// TIA Portal project "examen2" (V15.1)

(* hardware
DEVICE "S7-1200 station_1"  S7-1200 Station
   slot 0: "Rack_0"  S7-1200 Rack  Rack  V1.0
   slot 1: "03_BANDA"  CPU 1212C AC/DC/Rly  6ES7 212-1BE40-0XB0  V4.2
   slot 3: "AQ 1x12BIT_1"  AQ1 signal board  6ES7 232-4HA30-0XB0  V1.0
DEVICE "S7-1200 station_2"  S7-1200 Station
   slot 0: "Rack_0"  S7-1200 Rack  Rack  V1.0
   slot 1: "01_CONTROL"  CPU 1214C AC/DC/Rly  6ES7 214-1BG40-0XB0  V4.2
   slot 2: "DI 8/DQ 8x24VDC_1"  6ES7 223-1BH32-0XB0  V2.0
   slot 3: "AQ 1x12BIT_1"  AQ1 signal board  6ES7 232-4HA30-0XB0  V1.0
DEVICE "S7-1200 station_3"  S7-1200 Station
   slot 0: "Rack_0"  S7-1200 Rack  Rack  V1.0
   slot 1: "02_ALMACEN"  CPU 1214C AC/DC/Rly  6ES7 214-1BG40-0XB0  V4.2
   slot 2: "DI 8x24VDC/DQ 8xRelay_1"  SM 1223 DI8/DQ8 x relay  6ES7 223-1PH32-0XB0  V2.0
*)

// ===== PLC "03_BANDA"  CPU 1212C AC/DC/Rly =====

VAR_GLOBAL   // PLC tag table "Tabla de variables estándar"
   "START" AT %M1.0 : Bool;
   "STOP" AT %M1.1 : Bool;
   "MEM0" AT %M1.2 : Bool;
   "SEN1" AT %I0.3 : Bool;
   "METALCOUNTER" AT %MW10 : Int;
   "PLASTICCOUNTER" AT %MW12 : Int;
   "MEM4" AT %M1.3 : Bool;
   "MEM1" AT %M1.4 : Bool;
   "SEN4" AT %I0.6 : Bool;
   "MEM2" AT %M1.5 : Bool;
   "MEM3" AT %M1.6 : Bool;
   "SEN5" AT %I0.7 : Bool;
   "SEN2" AT %I0.4 : Bool;
   "MEM5" AT %M1.7 : Bool;
   "SEN3" AT %I0.5 : Bool;
   "MOTORBANDA" AT %Q0.0 : Bool;
   "DATARCVS" AT %MB2 : Byte;
   "DATASENDS" AT %MB3 : Byte;
   "Tag_1" AT %QW80 : Int;
   "SUM_ST" AT %MW8 : Int;
   "COUNTER_MEM" AT %M0.0 : Bool;
   "AVISO" AT %M0.1 : Bool;
   "System_Byte" AT %MB1001 : Byte;
   "FirstScan" AT %M1001.0 : Bool;
   "DiagStatusUpdate" AT %M1001.1 : Bool;
   "AlwaysTRUE" AT %M1001.2 : Bool;
   "AlwaysFALSE" AT %M1001.3 : Bool;
   "Clock_Byte" AT %MB1002 : Byte;
   "Clock_10Hz" AT %M1002.0 : Bool;
   "Clock_5Hz" AT %M1002.1 : Bool;
   "Clock_2.5Hz" AT %M1002.2 : Bool;
   "Clock_2Hz" AT %M1002.3 : Bool;
   "Clock_1.25Hz" AT %M1002.4 : Bool;
   "Clock_1Hz" AT %M1002.5 : Bool;
   "Clock_0.625Hz" AT %M1002.6 : Bool;
   "Clock_0.5Hz" AT %M1002.7 : Bool;
   "BYTEINALM" AT %MB4 : Byte;
   "ENDPROCESS" AT %M0.2 : Bool;
   "FIN" AT %M0.3 : Bool;
   "STATUS2SEND" AT %M0.4 : Bool;
   "BYTE2SEND" AT %MB5 : Byte;
   "DATASENDS2" AT %MB6 : Byte;
   "BIT0SUM" AT %M0.5 : Bool;
   "BIT1SUM" AT %M0.6 : Bool;
   "BIT2SUM" AT %M0.7 : Bool;
   "BIT3SUM" AT %M7.0 : Bool;
   "DATA2SENDC" AT %MB14 : Byte;
END_VAR

// folder: System blocks/Program resources

DATA_BLOCK "METALCOUNT"   // DB1
{ S7_Optimized_Access := 'TRUE' }
AUTHOR : Simatic
FAMILY : IEC
NAME : CNTR
VERSION : 1.0
// stored: InstanceOfName IEC_COUNTER
"IEC_COUNTER"
BEGIN
END_DATA_BLOCK

DATA_BLOCK "PLASTCOUNT"   // DB2
{ S7_Optimized_Access := 'TRUE' }
AUTHOR : Simatic
FAMILY : IEC
NAME : CNTR
VERSION : 1.0
// stored: InstanceOfName IEC_COUNTER
"IEC_COUNTER"
BEGIN
END_DATA_BLOCK

DATA_BLOCK "TIM1"   // DB3
{ S7_Optimized_Access := 'TRUE' }
AUTHOR : Simatic
FAMILY : IEC
NAME : IEC_TMR
VERSION : 1.0
// stored: InstanceOfName IEC_TIMER
"IEC_TIMER"
BEGIN
END_DATA_BLOCK

DATA_BLOCK "_03_BANDA_Receive_DB_1"   // DB4
{ S7_Optimized_Access := 'TRUE' }
AUTHOR : SIMATIC
FAMILY : MC7Plus
NAME : TC_IP_v4
VERSION : 1.0
// stored: InstanceOfName TCON_IP_v4
"TCON_IP_v4"
BEGIN
   ID := 1;
   InterfaceId := 64;
   LocalPort := 2000;
   RemoteAddress.ADDR[1] := 192;
   RemoteAddress.ADDR[2] := 168;
   RemoteAddress.ADDR[4] := 2;
END_DATA_BLOCK

DATA_BLOCK "_03_BANDA_Receive_DB"   // DB8
{ S7_Optimized_Access := 'TRUE' }
AUTHOR : SIMATIC
FAMILY : MC7Plus
NAME : TC_IP_v4
VERSION : 1.0
// stored: InstanceOfName TCON_IP_v4
"TCON_IP_v4"
BEGIN
   ID := 3;
   InterfaceId := 64;
   LocalPort := 2001;
   RemoteAddress.ADDR[1] := 192;
   RemoteAddress.ADDR[2] := 168;
   RemoteAddress.ADDR[4] := 1;
END_DATA_BLOCK

DATA_BLOCK "_03_BANDA_Send_DB"   // DB9
{ S7_Optimized_Access := 'TRUE' }
AUTHOR : SIMATIC
FAMILY : MC7Plus
NAME : TC_IP_v4
VERSION : 1.0
// stored: InstanceOfName TCON_IP_v4
"TCON_IP_v4"
BEGIN
   ID := 4;
   InterfaceId := 64;
   RemotePort := 2000;
   ActiveEstablished := true;
   RemoteAddress.ADDR[1] := 192;
   RemoteAddress.ADDR[2] := 168;
   RemoteAddress.ADDR[4] := 1;
END_DATA_BLOCK

DATA_BLOCK "TIMER3"   // DB10
{ S7_Optimized_Access := 'TRUE' }
AUTHOR : Simatic
FAMILY : IEC
NAME : IEC_TMR
VERSION : 1.0
// stored: InstanceOfName IEC_TIMER
"IEC_TIMER"
BEGIN
END_DATA_BLOCK

DATA_BLOCK "_03_BANDA_Send_DB_1"   // DB12
{ S7_Optimized_Access := 'TRUE' }
AUTHOR : SIMATIC
FAMILY : MC7Plus
NAME : TC_IP_v4
VERSION : 1.0
// stored: InstanceOfName TCON_IP_v4
"TCON_IP_v4"
BEGIN
   ID := 2;
   InterfaceId := 64;
   RemotePort := 2000;
   ActiveEstablished := true;
   RemoteAddress.ADDR[1] := 192;
   RemoteAddress.ADDR[2] := 168;
   RemoteAddress.ADDR[4] := 2;
END_DATA_BLOCK

DATA_BLOCK "_03_BANDA_Send_DB_3"   // DB16
{ S7_Optimized_Access := 'TRUE' }
AUTHOR : SIMATIC
FAMILY : MC7Plus
NAME : TC_IP_v4
VERSION : 1.0
// stored: InstanceOfName TCON_IP_v4
"TCON_IP_v4"
BEGIN
   ID := 6;
   InterfaceId := 64;
   RemotePort := 2002;
   ActiveEstablished := true;
   RemoteAddress.ADDR[1] := 192;
   RemoteAddress.ADDR[2] := 168;
   RemoteAddress.ADDR[4] := 1;
END_DATA_BLOCK

DATA_BLOCK "_03_BANDA_Send_DB_2"   // DB18
{ S7_Optimized_Access := 'TRUE' }
AUTHOR : SIMATIC
FAMILY : MC7Plus
NAME : TC_IP_v4
VERSION : 1.0
// stored: InstanceOfName TCON_IP_v4
"TCON_IP_v4"
BEGIN
   ID := 5;
   InterfaceId := 64;
   RemotePort := 2000;
   ActiveEstablished := true;
   RemoteAddress.ADDR[1] := 192;
   RemoteAddress.ADDR[2] := 168;
   RemoteAddress.ADDR[4] := 1;
END_DATA_BLOCK

// folder: (top level)

FUNCTION "CODER" : Void   // FC1, FBD
{ S7_Optimized_Access := 'TRUE' }
VERSION : 0.1
   VAR_INPUT
      BIT0 : Bool;
      BIT1 : Bool;
      BIT2 : Bool;
      BIT3 : Bool;
      BIT4 : Bool;
      BIT5 : Bool;
      BIT6 : Bool;
      BIT7 : Bool;
   END_VAR
   VAR_IN_OUT
      OUT : Byte;
   END_VAR
   VAR_TEMP
      MASK0 : Byte;
      MASK1 : Byte;
      MASK2 : Byte;
      MASK3 : Byte;
      MASK4 : Byte;
      MASK5 : Byte;
      MASK6 : Byte;
      MASK7 : Byte;
      MASK : Byte;
      MASK0N : Byte;
      MASK1N : Byte;
      MASK2N : Byte;
      MASK3N : Byte;
      MASK4N : Byte;
      MASK5N : Byte;
      MASK6N : Byte;
      MASK7N : Byte;
      MASKN : Byte;
   END_VAR
BEGIN

REGION Network 1
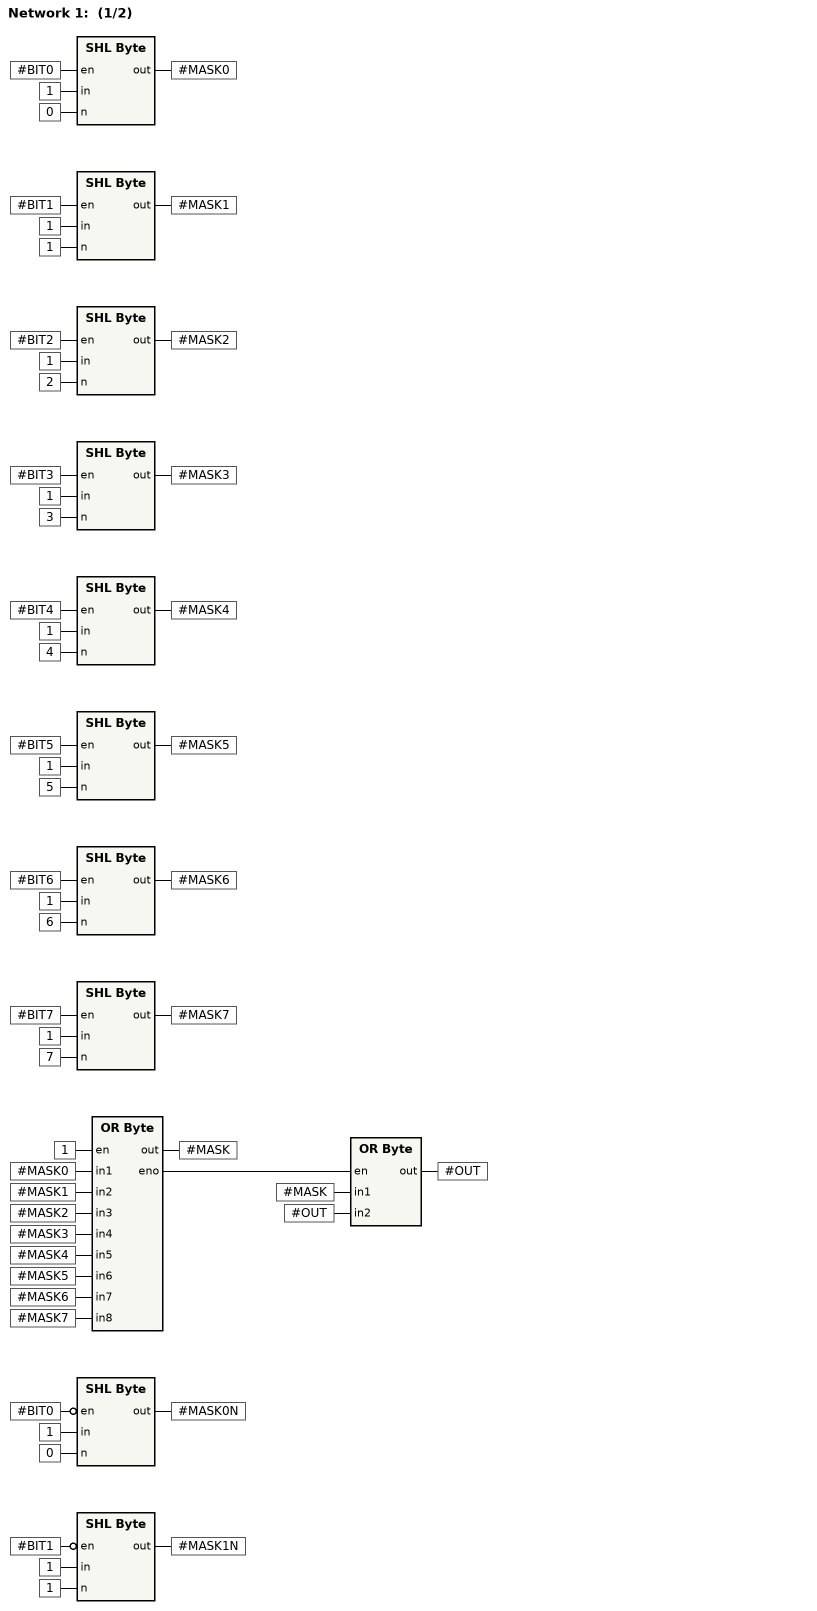
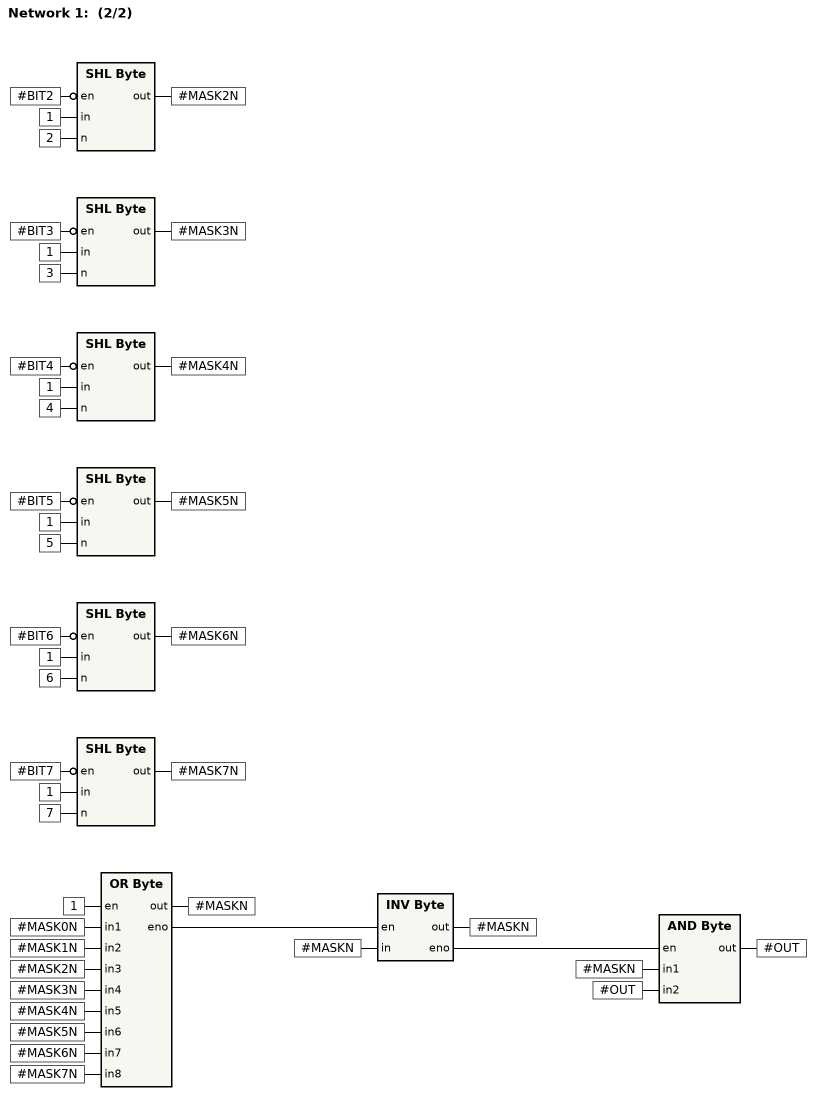
   IF #BIT0 THEN #MASK0 := SHL(IN := 1, N := 0); END_IF;
   IF #BIT1 THEN #MASK1 := SHL(IN := 1, N := 1); END_IF;
   IF #BIT2 THEN #MASK2 := SHL(IN := 1, N := 2); END_IF;
   IF #BIT3 THEN #MASK3 := SHL(IN := 1, N := 3); END_IF;
   IF #BIT4 THEN #MASK4 := SHL(IN := 1, N := 4); END_IF;
   IF #BIT5 THEN #MASK5 := SHL(IN := 1, N := 5); END_IF;
   IF #BIT6 THEN #MASK6 := SHL(IN := 1, N := 6); END_IF;
   IF #BIT7 THEN #MASK7 := SHL(IN := 1, N := 7); END_IF;
   IF 1 THEN
       #MASK := #MASK0 OR #MASK1 OR #MASK2 OR #MASK3 OR #MASK4 OR #MASK5 OR #MASK6 OR #MASK7;
       #OUT := #MASK OR #OUT;
   END_IF;
   IF NOT #BIT0 THEN #MASK0N := SHL(IN := 1, N := 0); END_IF;
   IF NOT #BIT1 THEN #MASK1N := SHL(IN := 1, N := 1); END_IF;
   IF NOT #BIT2 THEN #MASK2N := SHL(IN := 1, N := 2); END_IF;
   IF NOT #BIT3 THEN #MASK3N := SHL(IN := 1, N := 3); END_IF;
   IF NOT #BIT4 THEN #MASK4N := SHL(IN := 1, N := 4); END_IF;
   IF NOT #BIT5 THEN #MASK5N := SHL(IN := 1, N := 5); END_IF;
   IF NOT #BIT6 THEN #MASK6N := SHL(IN := 1, N := 6); END_IF;
   IF NOT #BIT7 THEN #MASK7N := SHL(IN := 1, N := 7); END_IF;
   IF 1 THEN
       #MASKN := #MASK0N OR #MASK1N OR #MASK2N OR #MASK3N OR #MASK4N OR #MASK5N OR #MASK6N OR #MASK7N;
       #MASKN := NOT #MASKN;
       #OUT := #MASKN AND #OUT;
   END_IF;
END_REGION
END_FUNCTION

FUNCTION "DECODER" : Void   // FC2, FBD
{ S7_Optimized_Access := 'TRUE' }
VERSION : 0.1
   VAR_INPUT
      INBYTE : Byte;
   END_VAR
   VAR_OUTPUT
      BIT0 : Bool;
      BIT1 : Bool;
      BIT2 : Bool;
      BIT3 : Bool;
      BIT4 : Bool;
      BIT5 : Bool;
      BIT6 : Bool;
      BIT7 : Bool;
   END_VAR
   VAR_TEMP
      MASK0 : Byte;
      MASK1 : Byte;
      MASK2 : Byte;
      MASK3 : Byte;
      MASK4 : Byte;
      MASK5 : Byte;
      MASK6 : Byte;
      MASK7 : Byte;
      OUTBIT0 : Byte;
      OUTBIT1 : Byte;
      OUTBIT2 : Byte;
      OUTBIT3 : Byte;
      OUTBIT4 : Byte;
      OUTBIT5 : Byte;
      OUTBIT6 : Byte;
      OUTBIT7 : Byte;
   END_VAR
BEGIN

REGION Network 1
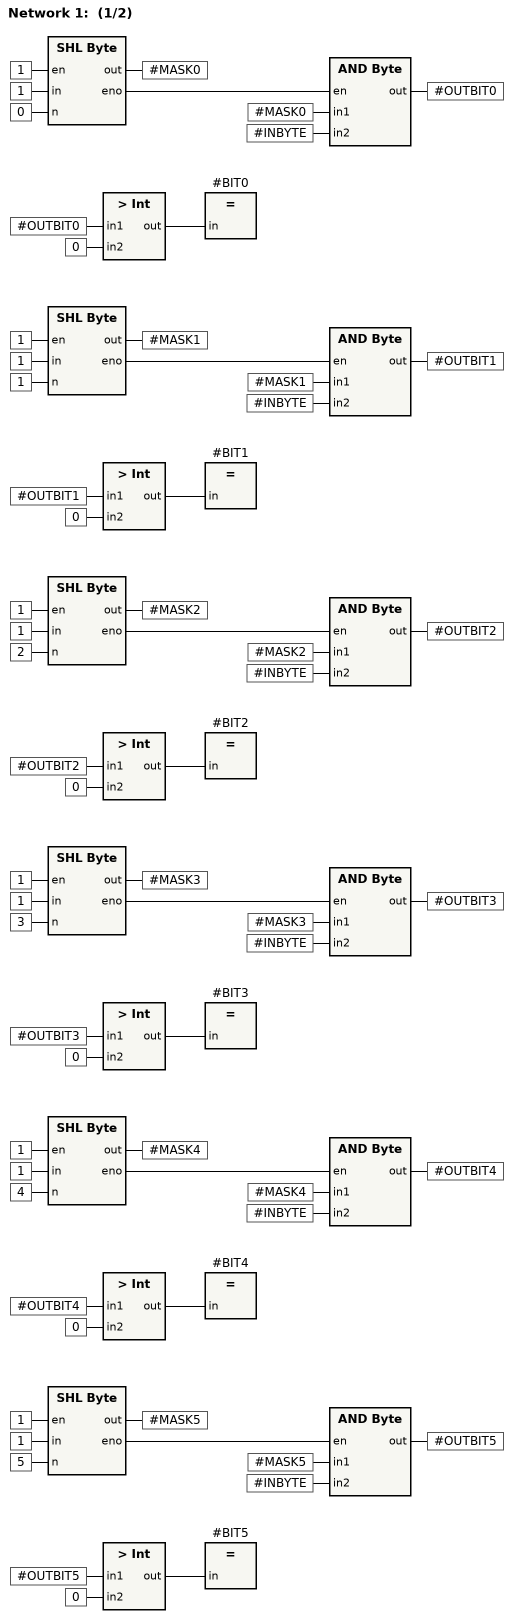
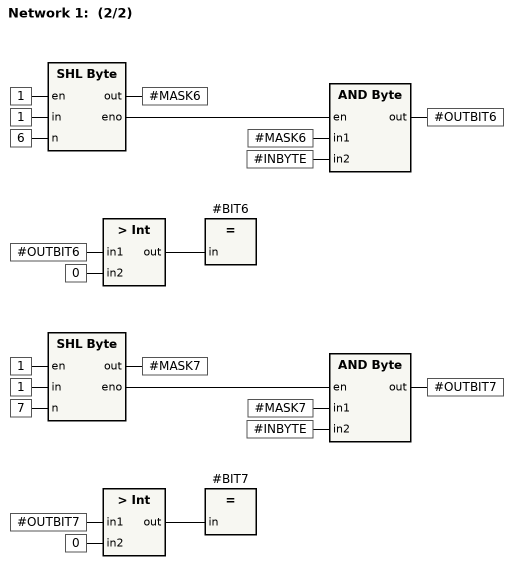
   IF 1 THEN
       #MASK0 := SHL(IN := 1, N := 0);
       #OUTBIT0 := #MASK0 AND #INBYTE;
   END_IF;
   #BIT0 := #OUTBIT0 > 0;
   IF 1 THEN
       #MASK1 := SHL(IN := 1, N := 1);
       #OUTBIT1 := #MASK1 AND #INBYTE;
   END_IF;
   #BIT1 := #OUTBIT1 > 0;
   IF 1 THEN
       #MASK2 := SHL(IN := 1, N := 2);
       #OUTBIT2 := #MASK2 AND #INBYTE;
   END_IF;
   #BIT2 := #OUTBIT2 > 0;
   IF 1 THEN
       #MASK3 := SHL(IN := 1, N := 3);
       #OUTBIT3 := #MASK3 AND #INBYTE;
   END_IF;
   #BIT3 := #OUTBIT3 > 0;
   IF 1 THEN
       #MASK4 := SHL(IN := 1, N := 4);
       #OUTBIT4 := #MASK4 AND #INBYTE;
   END_IF;
   #BIT4 := #OUTBIT4 > 0;
   IF 1 THEN
       #MASK5 := SHL(IN := 1, N := 5);
       #OUTBIT5 := #MASK5 AND #INBYTE;
   END_IF;
   #BIT5 := #OUTBIT5 > 0;
   IF 1 THEN
       #MASK6 := SHL(IN := 1, N := 6);
       #OUTBIT6 := #MASK6 AND #INBYTE;
   END_IF;
   #BIT6 := #OUTBIT6 > 0;
   IF 1 THEN
       #MASK7 := SHL(IN := 1, N := 7);
       #OUTBIT7 := #MASK7 AND #INBYTE;
   END_IF;
   #BIT7 := #OUTBIT7 > 0;
END_REGION
END_FUNCTION

FUNCTION "DecToBin" : Void   // FC3, FBD
{ S7_Optimized_Access := 'TRUE' }
VERSION : 0.1
   VAR_INPUT
      dec : Int;
   END_VAR
   VAR_OUTPUT
      bit0 : Bool;
      bit1 : Bool;
      bit2 : Bool;
      bit3 : Bool;
   END_VAR
   VAR_TEMP
      secdec : Int;
      thirdec : Int;
      quardec : Int;
      bit0s : Int;
      bit1s : Int;
      bit2s : Int;
      bit3s : Int;
   END_VAR
BEGIN

REGION Network 1
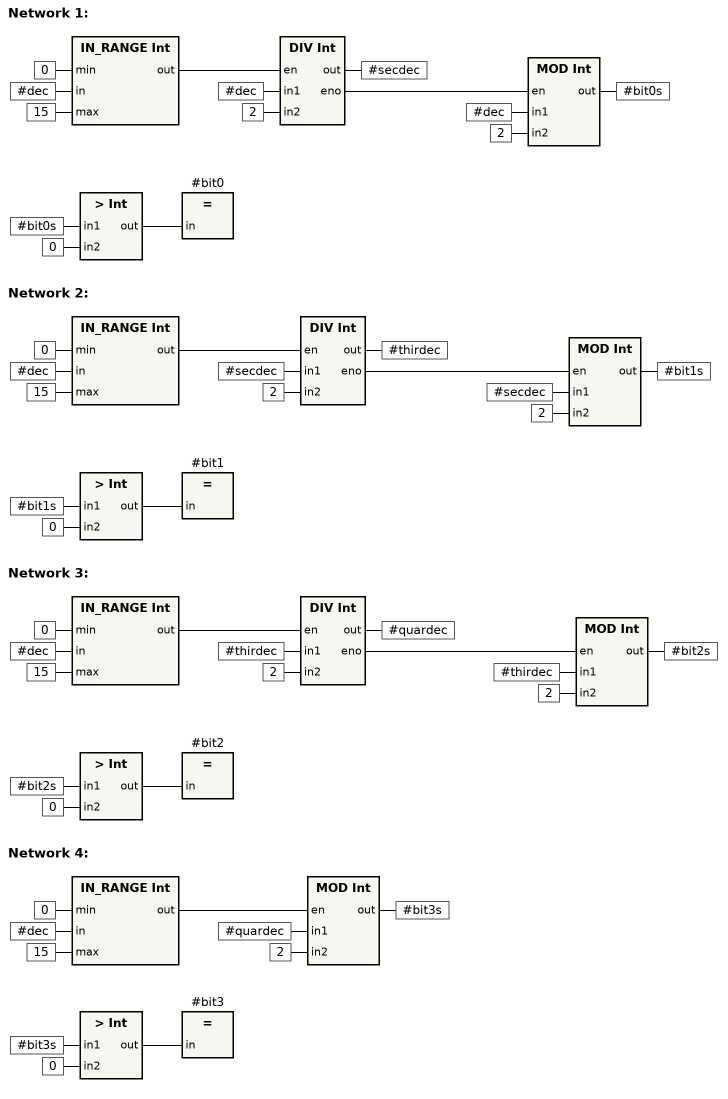
   IF (0 <= #dec) AND (#dec <= 15) THEN
       #secdec := #dec / 2;
       #bit0s := #dec MOD 2;
   END_IF;
   #bit0 := #bit0s > 0;
END_REGION

REGION Network 2
   IF (0 <= #dec) AND (#dec <= 15) THEN
       #thirdec := #secdec / 2;
       #bit1s := #secdec MOD 2;
   END_IF;
   #bit1 := #bit1s > 0;
END_REGION

REGION Network 3
   IF (0 <= #dec) AND (#dec <= 15) THEN
       #quardec := #thirdec / 2;
       #bit2s := #thirdec MOD 2;
   END_IF;
   #bit2 := #bit2s > 0;
END_REGION

REGION Network 4
   IF (0 <= #dec) AND (#dec <= 15) THEN #bit3s := #quardec MOD 2; END_IF;
   #bit3 := #bit3s > 0;
END_REGION
END_FUNCTION

FUNCTION "BinToDec" : Void   // FC4, FBD
{ S7_Optimized_Access := 'TRUE' }
VERSION : 0.1
   VAR_INPUT
      bit0 : Bool;
      bit1 : Bool;
      bit2 : Bool;
      bit3 : Bool;
   END_VAR
   VAR_OUTPUT
      decimal : Int;
   END_VAR
   VAR_TEMP
      dec0 : Int;
      dec1 : Int;
      dec2 : Int;
      dec3 : Int;
   END_VAR
BEGIN

REGION Network 1
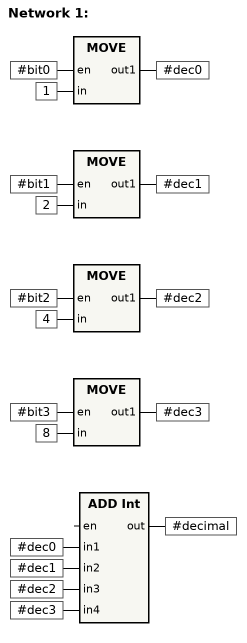
   IF #bit0 THEN #dec0 := 1; END_IF;
   IF #bit1 THEN #dec1 := 2; END_IF;
   IF #bit2 THEN #dec2 := 4; END_IF;
   IF #bit3 THEN #dec3 := 8; END_IF;
   #decimal := #dec0 + #dec1 + #dec2 + #dec3;
END_REGION
END_FUNCTION

ORGANIZATION_BLOCK "Main"   // OB1, LAD, ProgramCycle
TITLE = "Main Program Sweep (Cycle)" / "SLAVE_CONVEYOR_PLC"
{ S7_Optimized_Access := 'TRUE' }
VERSION : 0.1
   VAR_INPUT
      Initial_Call : Bool;   // Initial call of this OB
      Remanence : Bool;   // =True, if remanent data are available
   END_VAR
   VAR_TEMP
      SUMA : DInt;
      SUMA_ : Int;
      SUM_ : Int;
      BIT2 : Bool;
      BIT5 : Bool;
      BIT4 : Bool;
      BIT6 : Bool;
      BIT3 : Bool;
      BIT7 : Bool;
      MEM6 : Bool;
      MBIT0 : Bool;
      MBIT1 : Bool;
      MBIT2 : Bool;
      MBIT3 : Bool;
      MBIT4 : Bool;
      MBIT5 : Bool;
      MBIT6 : Bool;
   END_VAR
   VAR_TEMP   // added for the SCL form of the ladder/FBD networks
      _w1 : Bool;
   END_VAR
BEGIN

REGION Network 1: LOGIC_SEGMENT
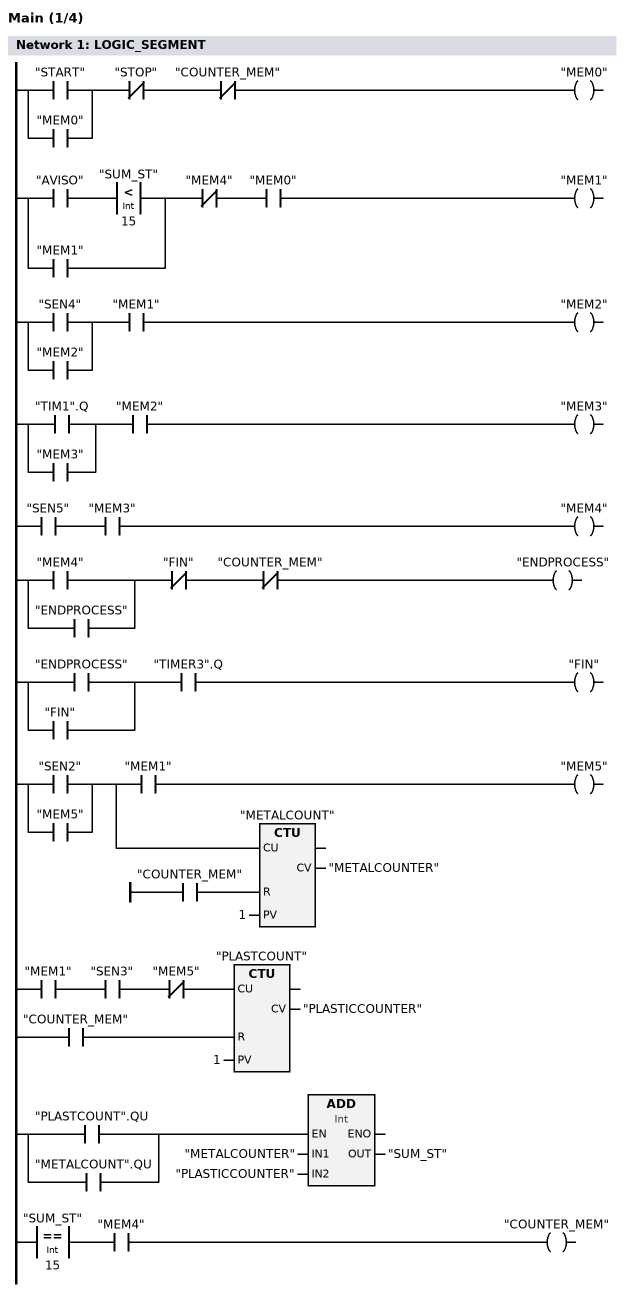
   "MEM0" := ("START" OR "MEM0") AND NOT "STOP" AND NOT "COUNTER_MEM";
   "MEM1" := (("AVISO" AND ("SUM_ST" < 15)) OR "MEM1") AND NOT "MEM4" AND "MEM0";
   "MEM2" := ("SEN4" OR "MEM2") AND "MEM1";
   "MEM3" := ("TIM1".Q OR "MEM3") AND "MEM2";
   "MEM4" := "SEN5" AND "MEM3";
   "ENDPROCESS" := ("MEM4" OR "ENDPROCESS") AND NOT "FIN" AND NOT "COUNTER_MEM";
   "FIN" := ("ENDPROCESS" OR "FIN") AND "TIMER3".Q;
   #_w1 := "SEN2" OR "MEM5";
   "MEM5" := #_w1 AND "MEM1";
   "METALCOUNT".CTU(CU := #_w1, R := "COUNTER_MEM", PV := 1, CV => "METALCOUNTER");
   "PLASTCOUNT".CTU(CU := "MEM1" AND "SEN3" AND NOT "MEM5", R := "COUNTER_MEM", PV := 1, CV => "PLASTICCOUNTER");
   IF "PLASTCOUNT".QU OR "METALCOUNT".QU THEN "SUM_ST" := "METALCOUNTER" + "PLASTICCOUNTER"; END_IF;
   "COUNTER_MEM" := ("SUM_ST" = 15) AND "MEM4";
END_REGION

REGION Network 2: MECHANICAL_SEGMENT
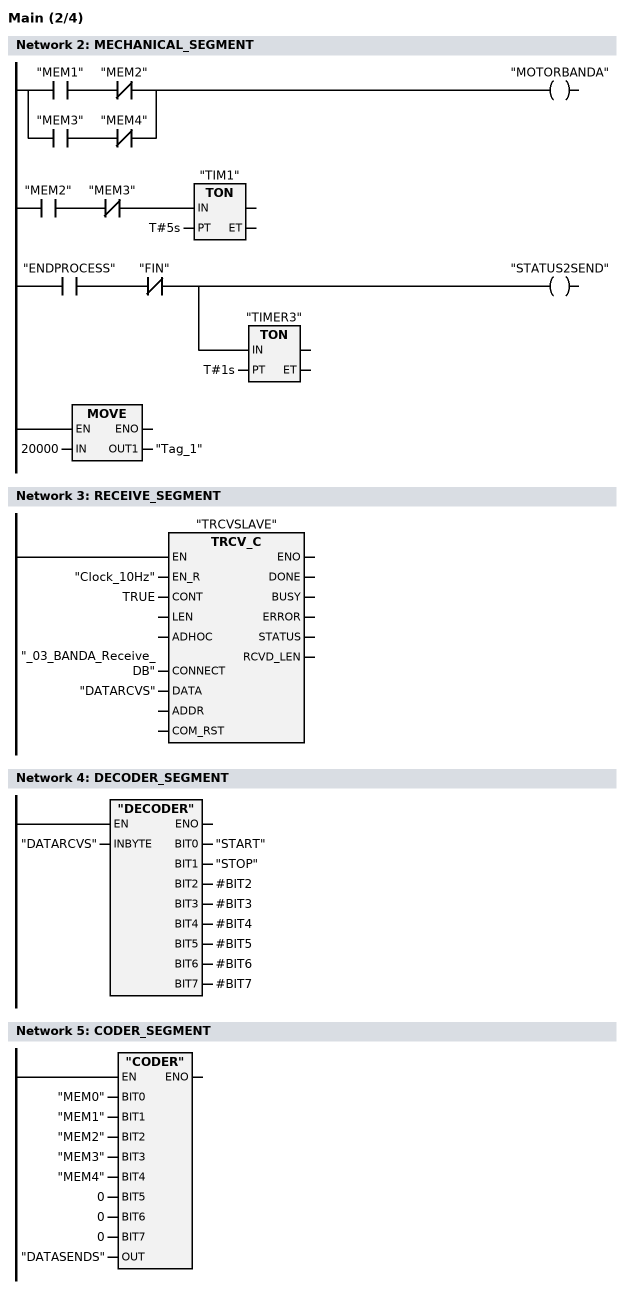
   "MOTORBANDA" := ("MEM1" AND NOT "MEM2") OR ("MEM3" AND NOT "MEM4");
   "TIM1".TON(IN := "MEM2" AND NOT "MEM3", PT := T#5s);
   "STATUS2SEND" := "ENDPROCESS" AND NOT "FIN";
   "TIMER3".TON(IN := "STATUS2SEND", PT := T#1s);
   "Tag_1" := 20000;
END_REGION

REGION Network 3: RECEIVE_SEGMENT
   "TRCVSLAVE"(EN_R := "Clock_10Hz", CONT := TRUE, CONNECT := "_03_BANDA_Receive_DB", DATA := "DATARCVS");   // TRCV_C
END_REGION

REGION Network 4: DECODER_SEGMENT
   RUNG wire#powerrail
      "DECODER"(INBYTE := "DATARCVS", BIT0 => "START", BIT1 => "STOP", BIT2 => #BIT2, BIT3 => #BIT3, BIT4 => #BIT4, BIT5 => #BIT5, BIT6 => #BIT6, BIT7 => #BIT7)
   END_RUNG
   // the same network as SCL:
   "DECODER"(INBYTE := "DATARCVS",
             BIT0 => "START",
             BIT1 => "STOP",
             BIT2 => #BIT2,
             BIT3 => #BIT3,
             BIT4 => #BIT4,
             BIT5 => #BIT5,
             BIT6 => #BIT6,
             BIT7 => #BIT7);
END_REGION

REGION Network 5: CODER_SEGMENT
   RUNG wire#powerrail
      "CODER"(BIT0 := "MEM0", BIT1 := "MEM1", BIT2 := "MEM2", BIT3 := "MEM3", BIT4 := "MEM4", BIT5 := 0, BIT6 := 0, BIT7 := 0, OUT := "DATASENDS")
   END_RUNG
   // the same network as SCL:
   "CODER"(BIT0 := "MEM0",
           BIT1 := "MEM1",
           BIT2 := "MEM2",
           BIT3 := "MEM3",
           BIT4 := "MEM4",
           BIT5 := 0,
           BIT6 := 0,
           BIT7 := 0,
           OUT := "DATASENDS");
END_REGION

REGION Network 6: SEND_SEGMENT
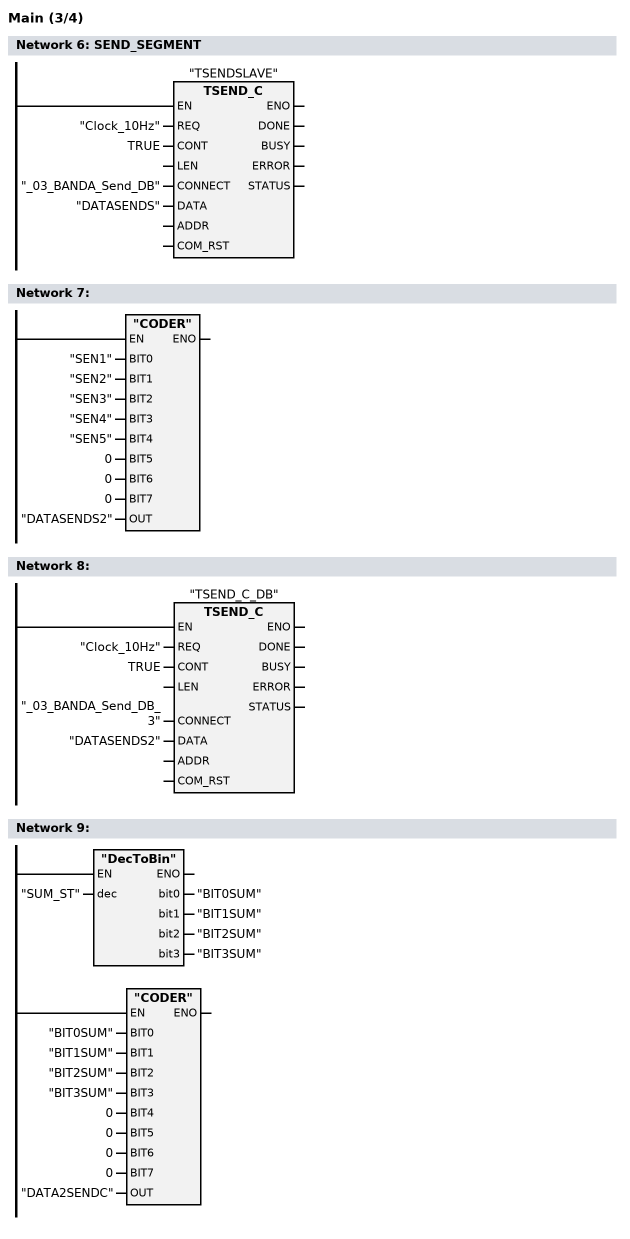
   "TSENDSLAVE"(REQ := "Clock_10Hz", CONT := TRUE, CONNECT := "_03_BANDA_Send_DB", DATA := "DATASENDS");   // TSEND_C
END_REGION

REGION Network 7
   RUNG wire#powerrail
      "CODER"(BIT0 := "SEN1", BIT1 := "SEN2", BIT2 := "SEN3", BIT3 := "SEN4", BIT4 := "SEN5", BIT5 := 0, BIT6 := 0, BIT7 := 0, OUT := "DATASENDS2")
   END_RUNG
   // the same network as SCL:
   "CODER"(BIT0 := "SEN1",
           BIT1 := "SEN2",
           BIT2 := "SEN3",
           BIT3 := "SEN4",
           BIT4 := "SEN5",
           BIT5 := 0,
           BIT6 := 0,
           BIT7 := 0,
           OUT := "DATASENDS2");
END_REGION

REGION Network 8
   "TSEND_C_DB"(REQ := "Clock_10Hz", CONT := TRUE, CONNECT := "_03_BANDA_Send_DB_3", DATA := "DATASENDS2");   // TSEND_C
END_REGION

REGION Network 9
   RUNG wire#powerrail
      "DecToBin"(dec := "SUM_ST", bit0 => "BIT0SUM", bit1 => "BIT1SUM", bit2 => "BIT2SUM", bit3 => "BIT3SUM")
   END_RUNG
   RUNG wire#powerrail
      "CODER"(BIT0 := "BIT0SUM", BIT1 := "BIT1SUM", BIT2 := "BIT2SUM", BIT3 := "BIT3SUM", BIT4 := 0, BIT5 := 0, BIT6 := 0, BIT7 := 0, OUT := "DATA2SENDC")
   END_RUNG
   // the same network as SCL:
   "DecToBin"(dec := "SUM_ST", bit0 => "BIT0SUM", bit1 => "BIT1SUM", bit2 => "BIT2SUM", bit3 => "BIT3SUM");
   "CODER"(BIT0 := "BIT0SUM",
           BIT1 := "BIT1SUM",
           BIT2 := "BIT2SUM",
           BIT3 := "BIT3SUM",
           BIT4 := 0,
           BIT5 := 0,
           BIT6 := 0,
           BIT7 := 0,
           OUT := "DATA2SENDC");
END_REGION

REGION Network 10
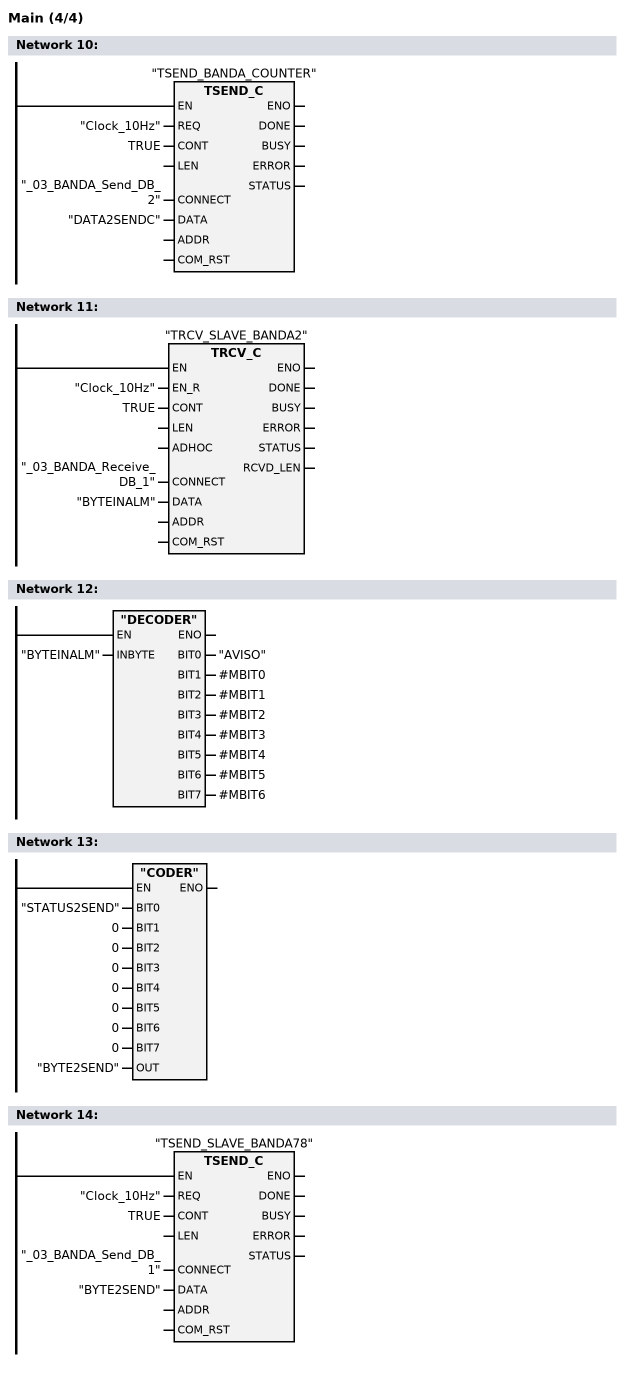
   "TSEND_BANDA_COUNTER"(REQ := "Clock_10Hz",   // TSEND_C
                         CONT := TRUE,
                         CONNECT := "_03_BANDA_Send_DB_2",
                         DATA := "DATA2SENDC");
END_REGION

REGION Network 11
   "TRCV_SLAVE_BANDA2"(EN_R := "Clock_10Hz",   // TRCV_C
                       CONT := TRUE,
                       CONNECT := "_03_BANDA_Receive_DB_1",
                       DATA := "BYTEINALM");
END_REGION

REGION Network 12
   RUNG wire#powerrail
      "DECODER"(INBYTE := "BYTEINALM", BIT0 => "AVISO", BIT1 => #MBIT0, BIT2 => #MBIT1, BIT3 => #MBIT2, BIT4 => #MBIT3, BIT5 => #MBIT4, BIT6 => #MBIT5, BIT7 => #MBIT6)
   END_RUNG
   // the same network as SCL:
   "DECODER"(INBYTE := "BYTEINALM",
             BIT0 => "AVISO",
             BIT1 => #MBIT0,
             BIT2 => #MBIT1,
             BIT3 => #MBIT2,
             BIT4 => #MBIT3,
             BIT5 => #MBIT4,
             BIT6 => #MBIT5,
             BIT7 => #MBIT6);
END_REGION

REGION Network 13
   RUNG wire#powerrail
      "CODER"(BIT0 := "STATUS2SEND", BIT1 := 0, BIT2 := 0, BIT3 := 0, BIT4 := 0, BIT5 := 0, BIT6 := 0, BIT7 := 0, OUT := "BYTE2SEND")
   END_RUNG
   // the same network as SCL:
   "CODER"(BIT0 := "STATUS2SEND",
           BIT1 := 0,
           BIT2 := 0,
           BIT3 := 0,
           BIT4 := 0,
           BIT5 := 0,
           BIT6 := 0,
           BIT7 := 0,
           OUT := "BYTE2SEND");
END_REGION

REGION Network 14
   "TSEND_SLAVE_BANDA78"(REQ := "Clock_10Hz",   // TSEND_C
                         CONT := TRUE,
                         CONNECT := "_03_BANDA_Send_DB_1",
                         DATA := "BYTE2SEND");
END_REGION
END_ORGANIZATION_BLOCK

// ===== PLC "01_CONTROL"  CPU 1214C AC/DC/Rly =====

VAR_GLOBAL   // PLC tag table "Tabla de variables estándar"
   "START" AT %I0.0 : Bool;
   "STOP" AT %I0.1 : Bool;
   "MEM0" AT %M1.0 : Bool;
   "DATASENDM" AT %MB1 : Byte;
   "MEM1" AT %M1.2 : Bool;
   "MEM2" AT %M1.3 : Bool;
   "GREEN" AT %Q8.5 : Bool;
   "MEM3" AT %M1.4 : Bool;
   "MEM4" AT %M1.5 : Bool;
   "ORANGE" AT %Q8.6 : Bool;
   "RED" AT %Q8.7 : Bool;
   "DATARCVM" AT %MB2 : Byte;
   "START2" AT %M3.0 : Bool;
   "SEN1" AT %M1.7 : Bool;
   "STOP2" AT %M0.0 : Bool;
   "TRY" AT %Q0.0 : Bool;
   "System_Byte" AT %MB10 : Byte;
   "FirstScan" AT %M10.0 : Bool;
   "DiagStatusUpdate" AT %M10.1 : Bool;
   "AlwaysTRUE" AT %M10.2 : Bool;
   "AlwaysFALSE" AT %M10.3 : Bool;
   "Clock_Byte" AT %MB11 : Byte;
   "Clock_10Hz" AT %M11.0 : Bool;
   "Clock_5Hz" AT %M11.1 : Bool;
   "Clock_2.5Hz" AT %M11.2 : Bool;
   "Clock_2Hz" AT %M11.3 : Bool;
   "Clock_1.25Hz" AT %M11.4 : Bool;
   "Clock_1Hz" AT %M11.5 : Bool;
   "Clock_0.625Hz" AT %M11.6 : Bool;
   "Clock_0.5Hz" AT %M11.7 : Bool;
   "SEN4" AT %M0.1 : Bool;
   "SEN3" AT %M0.2 : Bool;
   "SEN2" AT %M0.3 : Bool;
   "SEN5" AT %M0.4 : Bool;
   "COUNT1" AT %MB7 : Byte;
   "DATARCVS" AT %MB6 : Byte;
END_VAR

DATA_BLOCK "Data_block_1"   // DB2
{ S7_Optimized_Access := 'FALSE' }
VERSION : 0.1
   VAR
      BYTE0 : Byte;
      BYTE1 : Byte;
      BYTE2 : Byte;
      BYTE4 : Byte;
   END_VAR
BEGIN
END_DATA_BLOCK

// folder: System blocks/Program resources

DATA_BLOCK "_01_CONTROL_Receive_DB_1"   // DB3
{ S7_Optimized_Access := 'TRUE' }
AUTHOR : SIMATIC
FAMILY : MC7Plus
NAME : TC_IP_v4
VERSION : 1.0
// stored: InstanceOfName TCON_IP_v4
"TCON_IP_v4"
BEGIN
   ID := 1;
   InterfaceId := 64;
   LocalPort := 2000;
   RemoteAddress.ADDR[1] := 192;
   RemoteAddress.ADDR[2] := 168;
   RemoteAddress.ADDR[4] := 3;
END_DATA_BLOCK

DATA_BLOCK "_01_CONTROL_Send_DB"   // DB5
{ S7_Optimized_Access := 'TRUE' }
AUTHOR : SIMATIC
FAMILY : MC7Plus
NAME : TC_IP_v4
VERSION : 1.0
// stored: InstanceOfName TCON_IP_v4
"TCON_IP_v4"
BEGIN
   ID := 3;
   InterfaceId := 64;
   RemotePort := 2001;
   ActiveEstablished := true;
   RemoteAddress.ADDR[1] := 192;
   RemoteAddress.ADDR[2] := 168;
   RemoteAddress.ADDR[4] := 3;
END_DATA_BLOCK

DATA_BLOCK "_01_CONTROL_Receive_DB"   // DB6
{ S7_Optimized_Access := 'TRUE' }
AUTHOR : SIMATIC
FAMILY : MC7Plus
NAME : TC_IP_v4
VERSION : 1.0
// stored: InstanceOfName TCON_IP_v4
"TCON_IP_v4"
BEGIN
   ID := 4;
   InterfaceId := 64;
   LocalPort := 2000;
   RemoteAddress.ADDR[1] := 192;
   RemoteAddress.ADDR[2] := 168;
   RemoteAddress.ADDR[4] := 3;
END_DATA_BLOCK

DATA_BLOCK "_01_CONTROL_Receive_DB_2"   // DB7
{ S7_Optimized_Access := 'TRUE' }
AUTHOR : SIMATIC
FAMILY : MC7Plus
NAME : TC_IP_v4
VERSION : 1.0
// stored: InstanceOfName TCON_IP_v4
"TCON_IP_v4"
BEGIN
   ID := 2;
   InterfaceId := 64;
   LocalPort := 2002;
   RemoteAddress.ADDR[1] := 192;
   RemoteAddress.ADDR[2] := 168;
   RemoteAddress.ADDR[4] := 3;
END_DATA_BLOCK

// folder: (top level)

FUNCTION "CODER" : Void   // FC1, FBD
{ S7_Optimized_Access := 'TRUE' }
VERSION : 0.1
   VAR_INPUT
      BIT0 : Bool;
      BIT1 : Bool;
      BIT2 : Bool;
      BIT3 : Bool;
      BIT4 : Bool;
      BIT5 : Bool;
      BIT6 : Bool;
      BIT7 : Bool;
   END_VAR
   VAR_IN_OUT
      OUT : Byte;
   END_VAR
   VAR_TEMP
      MASK0 : Byte;
      MASK1 : Byte;
      MASK2 : Byte;
      MASK3 : Byte;
      MASK4 : Byte;
      MASK5 : Byte;
      MASK6 : Byte;
      MASK7 : Byte;
      MASK : Byte;
      MASK0N : Byte;
      MASK1N : Byte;
      MASK2N : Byte;
      MASK3N : Byte;
      MASK4N : Byte;
      MASK5N : Byte;
      MASK6N : Byte;
      MASK7N : Byte;
      MASKN : Byte;
   END_VAR
BEGIN

REGION Network 1
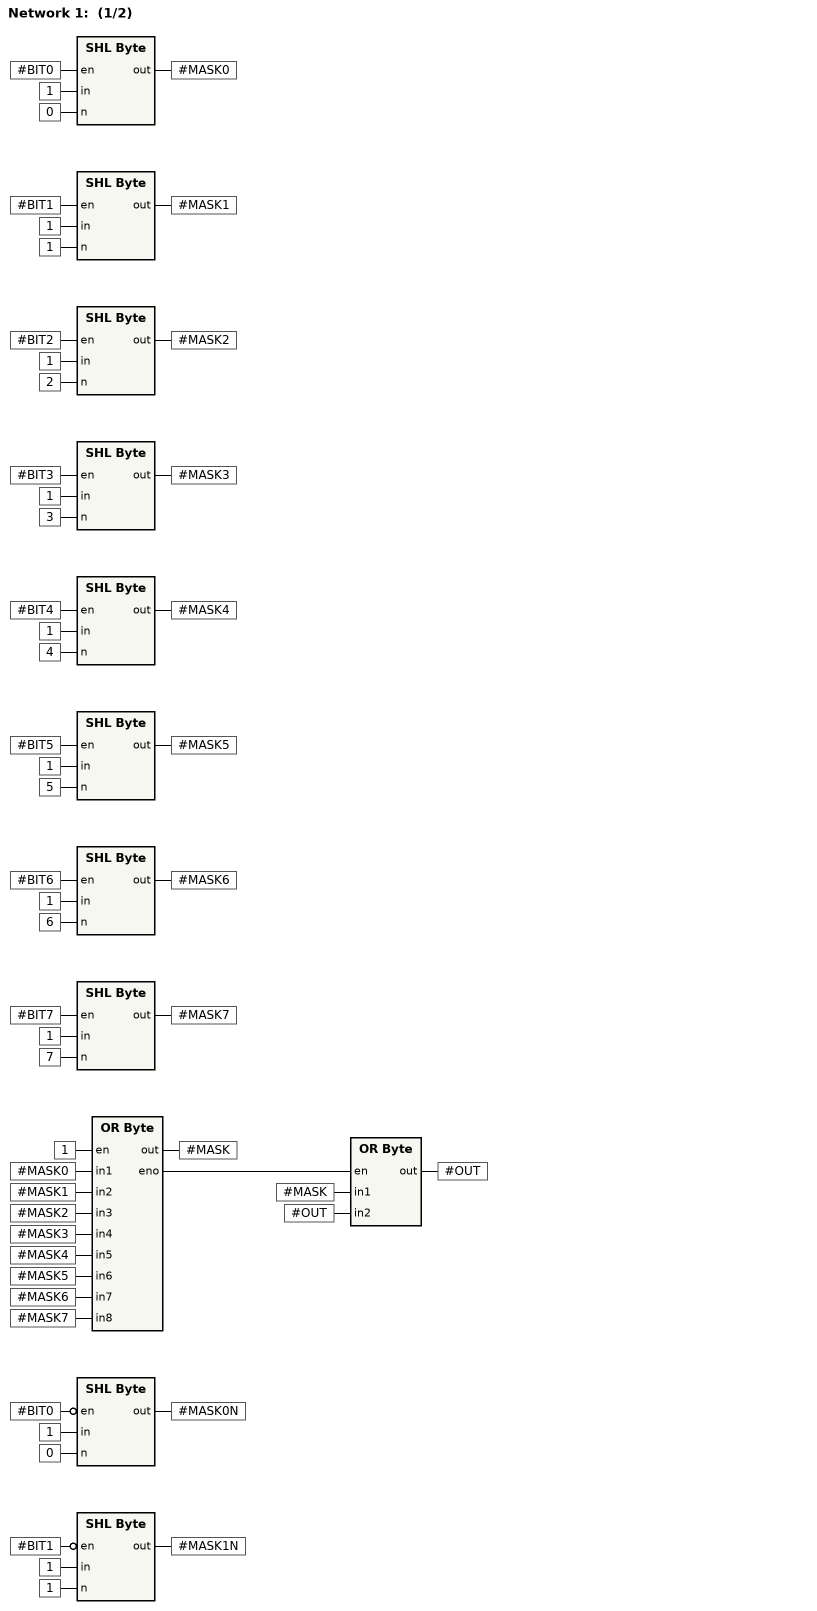
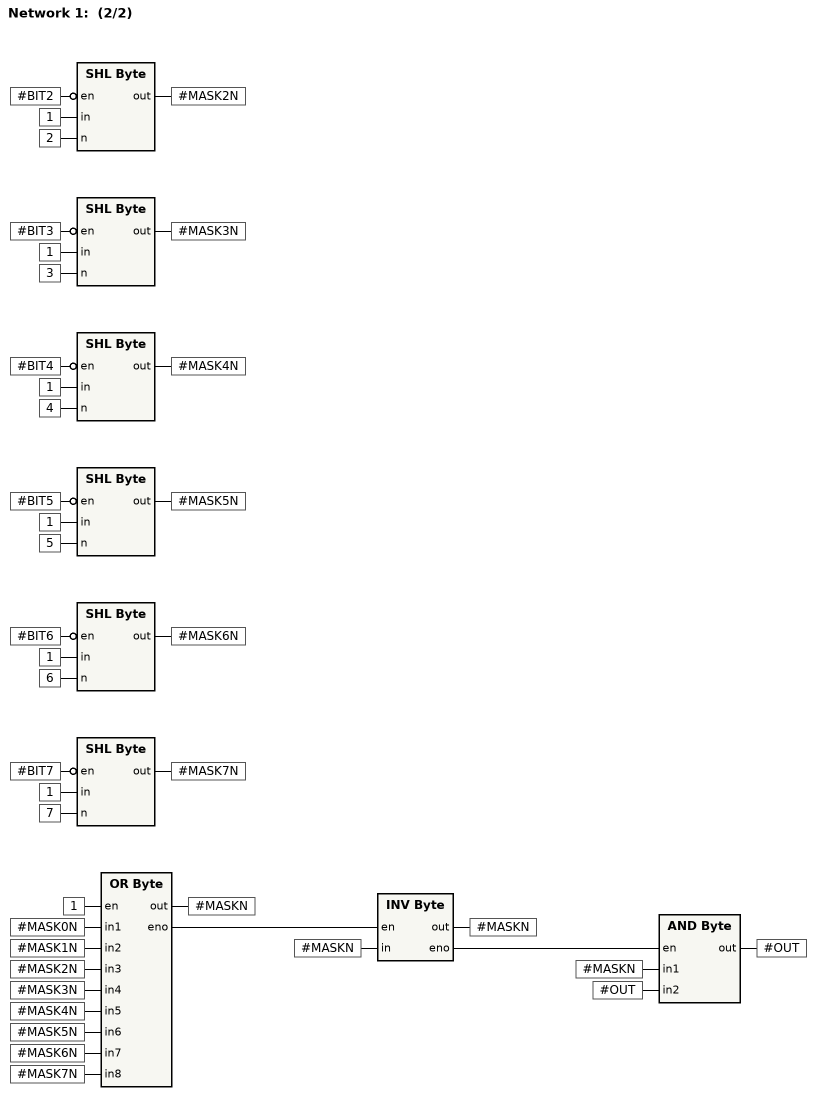
   IF #BIT0 THEN #MASK0 := SHL(IN := 1, N := 0); END_IF;
   IF #BIT1 THEN #MASK1 := SHL(IN := 1, N := 1); END_IF;
   IF #BIT2 THEN #MASK2 := SHL(IN := 1, N := 2); END_IF;
   IF #BIT3 THEN #MASK3 := SHL(IN := 1, N := 3); END_IF;
   IF #BIT4 THEN #MASK4 := SHL(IN := 1, N := 4); END_IF;
   IF #BIT5 THEN #MASK5 := SHL(IN := 1, N := 5); END_IF;
   IF #BIT6 THEN #MASK6 := SHL(IN := 1, N := 6); END_IF;
   IF #BIT7 THEN #MASK7 := SHL(IN := 1, N := 7); END_IF;
   IF 1 THEN
       #MASK := #MASK0 OR #MASK1 OR #MASK2 OR #MASK3 OR #MASK4 OR #MASK5 OR #MASK6 OR #MASK7;
       #OUT := #MASK OR #OUT;
   END_IF;
   IF NOT #BIT0 THEN #MASK0N := SHL(IN := 1, N := 0); END_IF;
   IF NOT #BIT1 THEN #MASK1N := SHL(IN := 1, N := 1); END_IF;
   IF NOT #BIT2 THEN #MASK2N := SHL(IN := 1, N := 2); END_IF;
   IF NOT #BIT3 THEN #MASK3N := SHL(IN := 1, N := 3); END_IF;
   IF NOT #BIT4 THEN #MASK4N := SHL(IN := 1, N := 4); END_IF;
   IF NOT #BIT5 THEN #MASK5N := SHL(IN := 1, N := 5); END_IF;
   IF NOT #BIT6 THEN #MASK6N := SHL(IN := 1, N := 6); END_IF;
   IF NOT #BIT7 THEN #MASK7N := SHL(IN := 1, N := 7); END_IF;
   IF 1 THEN
       #MASKN := #MASK0N OR #MASK1N OR #MASK2N OR #MASK3N OR #MASK4N OR #MASK5N OR #MASK6N OR #MASK7N;
       #MASKN := NOT #MASKN;
       #OUT := #MASKN AND #OUT;
   END_IF;
END_REGION
END_FUNCTION

FUNCTION "DECODER" : Void   // FC2, FBD
{ S7_Optimized_Access := 'TRUE' }
VERSION : 0.1
   VAR_INPUT
      INBYTE : Byte;
   END_VAR
   VAR_OUTPUT
      BIT0 : Bool;
      BIT1 : Bool;
      BIT2 : Bool;
      BIT3 : Bool;
      BIT4 : Bool;
      BIT5 : Bool;
      BIT6 : Bool;
      BIT7 : Bool;
   END_VAR
   VAR_TEMP
      MASK0 : Byte;
      MASK1 : Byte;
      MASK2 : Byte;
      MASK3 : Byte;
      MASK4 : Byte;
      MASK5 : Byte;
      MASK6 : Byte;
      MASK7 : Byte;
      OUTBIT0 : Byte;
      OUTBIT1 : Byte;
      OUTBIT2 : Byte;
      OUTBIT3 : Byte;
      OUTBIT4 : Byte;
      OUTBIT5 : Byte;
      OUTBIT6 : Byte;
      OUTBIT7 : Byte;
   END_VAR
BEGIN

REGION Network 1
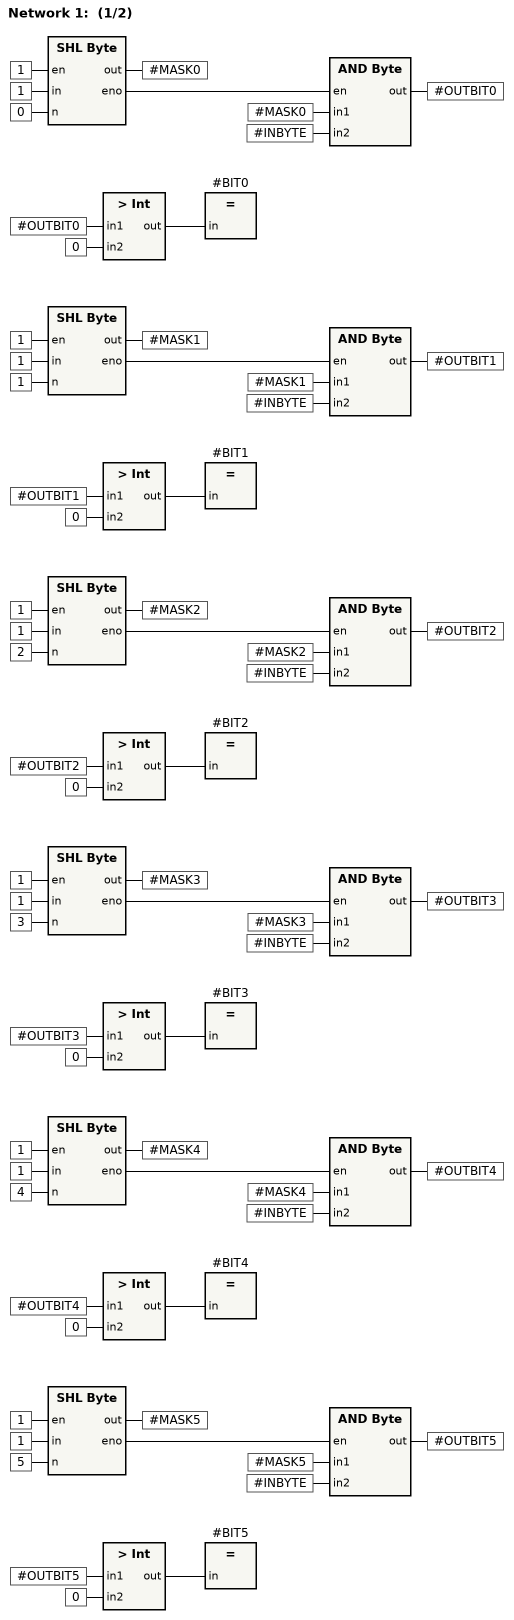
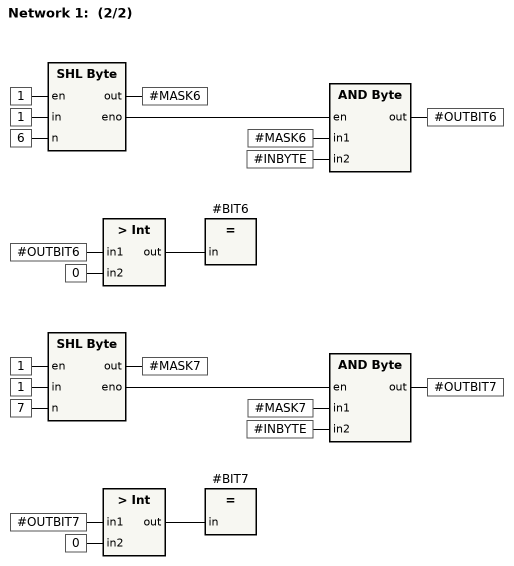
   IF 1 THEN
       #MASK0 := SHL(IN := 1, N := 0);
       #OUTBIT0 := #MASK0 AND #INBYTE;
   END_IF;
   #BIT0 := #OUTBIT0 > 0;
   IF 1 THEN
       #MASK1 := SHL(IN := 1, N := 1);
       #OUTBIT1 := #MASK1 AND #INBYTE;
   END_IF;
   #BIT1 := #OUTBIT1 > 0;
   IF 1 THEN
       #MASK2 := SHL(IN := 1, N := 2);
       #OUTBIT2 := #MASK2 AND #INBYTE;
   END_IF;
   #BIT2 := #OUTBIT2 > 0;
   IF 1 THEN
       #MASK3 := SHL(IN := 1, N := 3);
       #OUTBIT3 := #MASK3 AND #INBYTE;
   END_IF;
   #BIT3 := #OUTBIT3 > 0;
   IF 1 THEN
       #MASK4 := SHL(IN := 1, N := 4);
       #OUTBIT4 := #MASK4 AND #INBYTE;
   END_IF;
   #BIT4 := #OUTBIT4 > 0;
   IF 1 THEN
       #MASK5 := SHL(IN := 1, N := 5);
       #OUTBIT5 := #MASK5 AND #INBYTE;
   END_IF;
   #BIT5 := #OUTBIT5 > 0;
   IF 1 THEN
       #MASK6 := SHL(IN := 1, N := 6);
       #OUTBIT6 := #MASK6 AND #INBYTE;
   END_IF;
   #BIT6 := #OUTBIT6 > 0;
   IF 1 THEN
       #MASK7 := SHL(IN := 1, N := 7);
       #OUTBIT7 := #MASK7 AND #INBYTE;
   END_IF;
   #BIT7 := #OUTBIT7 > 0;
END_REGION
END_FUNCTION

FUNCTION "DecToBin" : Void   // FC3, FBD
{ S7_Optimized_Access := 'TRUE' }
VERSION : 0.1
   VAR_INPUT
      dec : Int;
   END_VAR
   VAR_OUTPUT
      bit0 : Bool;
      bit1 : Bool;
      bit2 : Bool;
      bit3 : Bool;
   END_VAR
   VAR_TEMP
      secdec : Int;
      thirdec : Int;
      quardec : Int;
      bit0s : Int;
      bit1s : Int;
      bit2s : Int;
      bit3s : Int;
   END_VAR
BEGIN

REGION Network 1
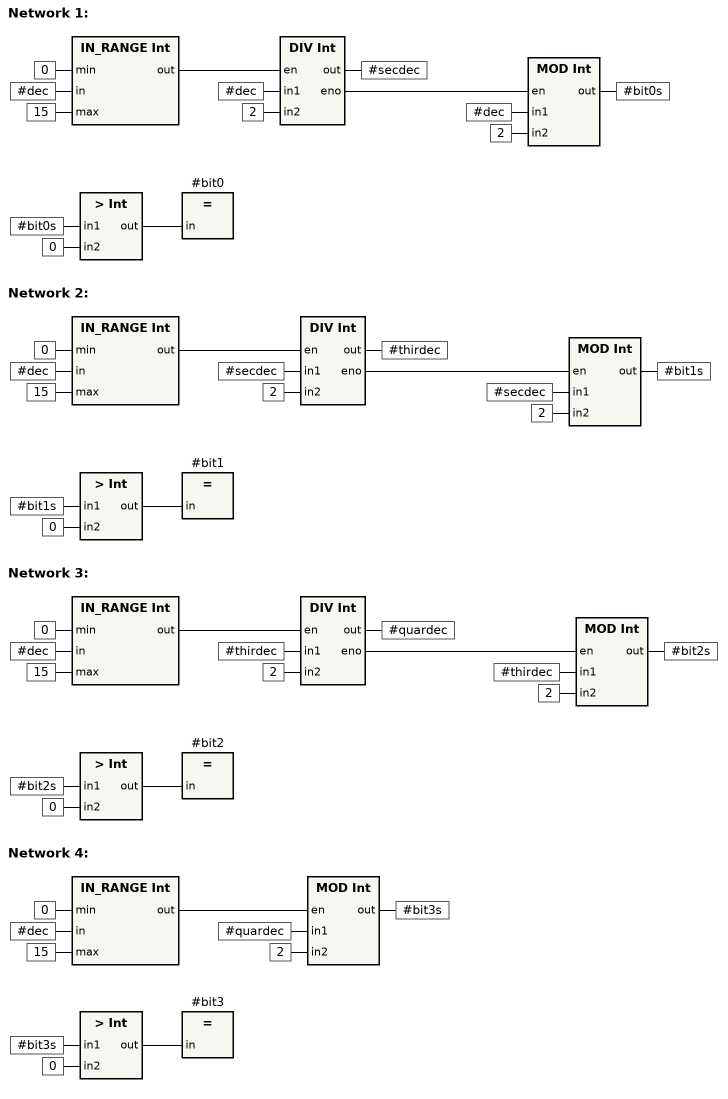
   IF (0 <= #dec) AND (#dec <= 15) THEN
       #secdec := #dec / 2;
       #bit0s := #dec MOD 2;
   END_IF;
   #bit0 := #bit0s > 0;
END_REGION

REGION Network 2
   IF (0 <= #dec) AND (#dec <= 15) THEN
       #thirdec := #secdec / 2;
       #bit1s := #secdec MOD 2;
   END_IF;
   #bit1 := #bit1s > 0;
END_REGION

REGION Network 3
   IF (0 <= #dec) AND (#dec <= 15) THEN
       #quardec := #thirdec / 2;
       #bit2s := #thirdec MOD 2;
   END_IF;
   #bit2 := #bit2s > 0;
END_REGION

REGION Network 4
   IF (0 <= #dec) AND (#dec <= 15) THEN #bit3s := #quardec MOD 2; END_IF;
   #bit3 := #bit3s > 0;
END_REGION
END_FUNCTION

FUNCTION "BinToDec" : Void   // FC4, FBD
{ S7_Optimized_Access := 'TRUE' }
VERSION : 0.1
   VAR_INPUT
      bit0 : Bool;
      bit1 : Bool;
      bit2 : Bool;
      bit3 : Bool;
   END_VAR
   VAR_OUTPUT
      decimal : Int;
   END_VAR
   VAR_TEMP
      dec0 : Int;
      dec1 : Int;
      dec2 : Int;
      dec3 : Int;
   END_VAR
BEGIN

REGION Network 1
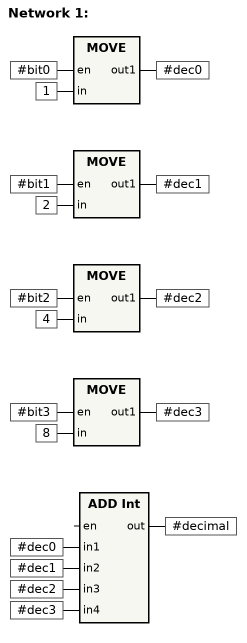
   IF #bit0 THEN #dec0 := 1; END_IF;
   IF #bit1 THEN #dec1 := 2; END_IF;
   IF #bit2 THEN #dec2 := 4; END_IF;
   IF #bit3 THEN #dec3 := 8; END_IF;
   #decimal := #dec0 + #dec1 + #dec2 + #dec3;
END_REGION
END_FUNCTION

ORGANIZATION_BLOCK "Main"   // OB1, LAD, ProgramCycle
TITLE = "Main Program Sweep (Cycle)" / "MASTER_PLC"
{ S7_Optimized_Access := 'TRUE' }
VERSION : 0.1
   VAR_INPUT
      Initial_Call : Bool;   // Initial call of this OB
      Remanence : Bool;   // =True, if remanent data are available
   END_VAR
   VAR_TEMP
      MEM6 : Bool;
      MEM5 : Bool;
      MEM7 : Bool;
      MEM8 : Bool;
      SEN6 : Bool;
      SEN7 : Bool;
      SEN8 : Bool;
   END_VAR
BEGIN

REGION Network 1: LOGIC_SEGMENT
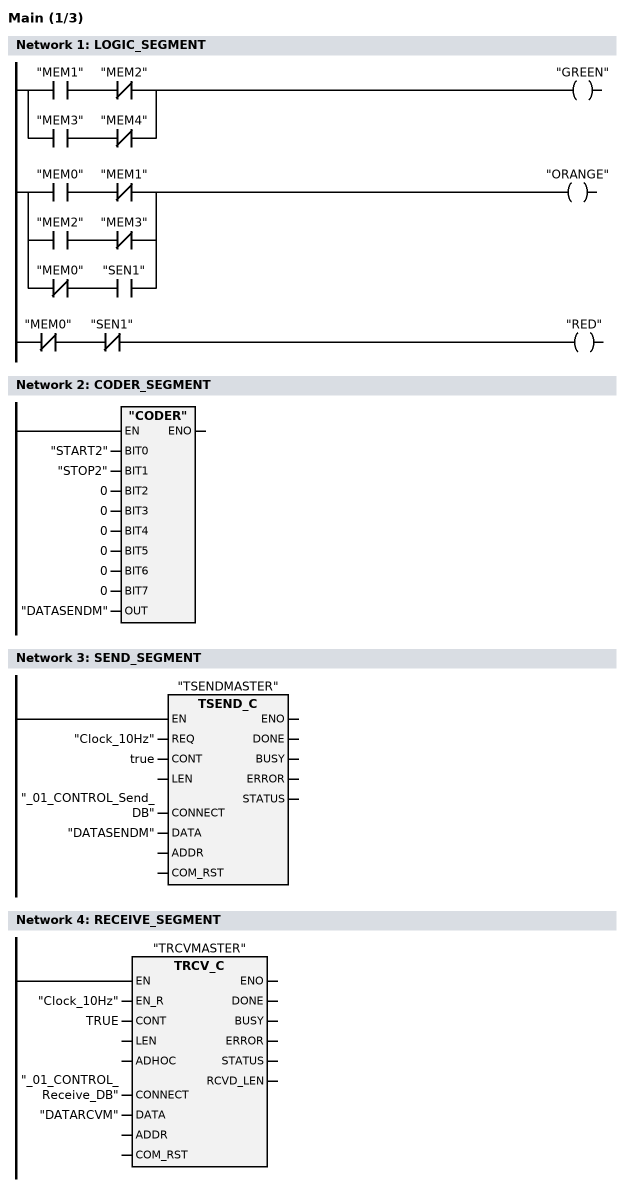
   RUNG wire#powerrail
      Contact( "MEM1" )
      I_Contact( "MEM2" )
      wire#w1
      Coil( "GREEN" )
   END_RUNG
   RUNG wire#powerrail
      Contact( "MEM3" )
      I_Contact( "MEM4" )
   END_RUNG wire#w1
   RUNG wire#powerrail
      Contact( "MEM0" )
      I_Contact( "MEM1" )
      wire#w2
      Coil( "ORANGE" )
   END_RUNG
   RUNG wire#powerrail
      Contact( "MEM2" )
      I_Contact( "MEM3" )
   END_RUNG wire#w2
   RUNG wire#powerrail
      I_Contact( "MEM0" )
      Contact( "SEN1" )
   END_RUNG wire#w2
   RUNG wire#powerrail
      I_Contact( "MEM0" )
      I_Contact( "SEN1" )
      Coil( "RED" )
   END_RUNG
   // the same network as SCL:
   "GREEN" := ("MEM1" AND NOT "MEM2") OR ("MEM3" AND NOT "MEM4");
   "ORANGE" := ("MEM0" AND NOT "MEM1") OR ("MEM2" AND NOT "MEM3") OR (NOT "MEM0" AND "SEN1");
   "RED" := NOT "MEM0" AND NOT "SEN1";
END_REGION

REGION Network 2: CODER_SEGMENT
   RUNG wire#powerrail
      "CODER"(BIT0 := "START2", BIT1 := "STOP2", BIT2 := 0, BIT3 := 0, BIT4 := 0, BIT5 := 0, BIT6 := 0, BIT7 := 0, OUT := "DATASENDM")
   END_RUNG
   // the same network as SCL:
   "CODER"(BIT0 := "START2",
           BIT1 := "STOP2",
           BIT2 := 0,
           BIT3 := 0,
           BIT4 := 0,
           BIT5 := 0,
           BIT6 := 0,
           BIT7 := 0,
           OUT := "DATASENDM");
END_REGION

REGION Network 3: SEND_SEGMENT
   "TSENDMASTER"(REQ := "Clock_10Hz", CONT := true, CONNECT := "_01_CONTROL_Send_DB", DATA := "DATASENDM");   // TSEND_C
END_REGION

REGION Network 4: RECEIVE_SEGMENT
   "TRCVMASTER"(EN_R := "Clock_10Hz", CONT := TRUE, CONNECT := "_01_CONTROL_Receive_DB", DATA := "DATARCVM");   // TRCV_C
END_REGION

REGION Network 5: DECODER_SEGMENT
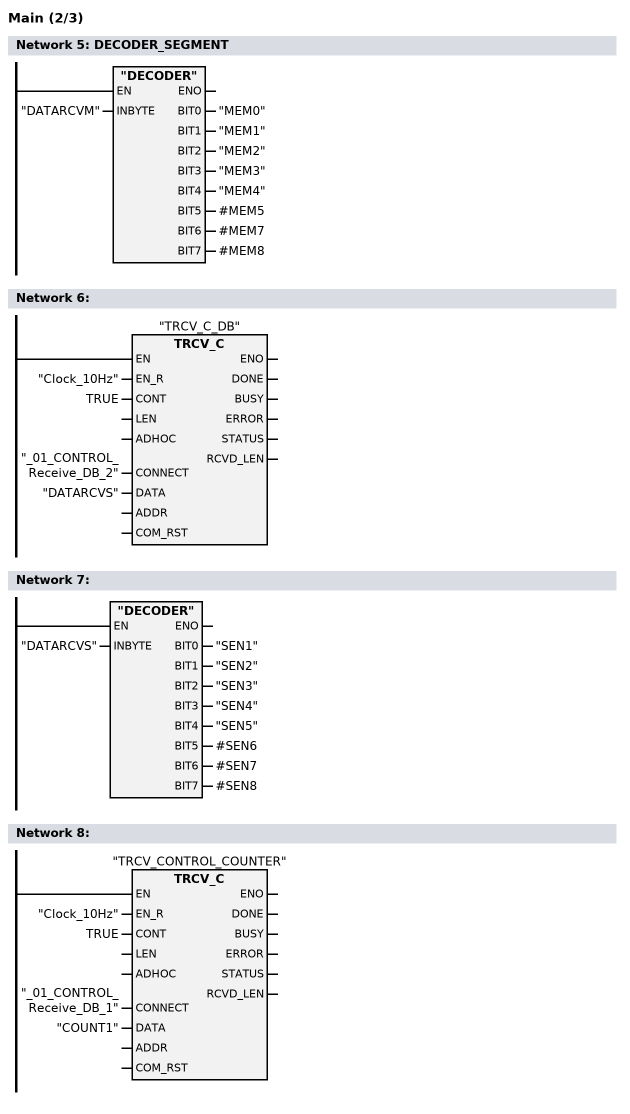
   RUNG wire#powerrail
      "DECODER"(INBYTE := "DATARCVM", BIT0 => "MEM0", BIT1 => "MEM1", BIT2 => "MEM2", BIT3 => "MEM3", BIT4 => "MEM4", BIT5 => #MEM5, BIT6 => #MEM7, BIT7 => #MEM8)
   END_RUNG
   // the same network as SCL:
   "DECODER"(INBYTE := "DATARCVM",
             BIT0 => "MEM0",
             BIT1 => "MEM1",
             BIT2 => "MEM2",
             BIT3 => "MEM3",
             BIT4 => "MEM4",
             BIT5 => #MEM5,
             BIT6 => #MEM7,
             BIT7 => #MEM8);
END_REGION

REGION Network 6
   "TRCV_C_DB"(EN_R := "Clock_10Hz", CONT := TRUE, CONNECT := "_01_CONTROL_Receive_DB_2", DATA := "DATARCVS");   // TRCV_C
END_REGION

REGION Network 7
   RUNG wire#powerrail
      "DECODER"(INBYTE := "DATARCVS", BIT0 => "SEN1", BIT1 => "SEN2", BIT2 => "SEN3", BIT3 => "SEN4", BIT4 => "SEN5", BIT5 => #SEN6, BIT6 => #SEN7, BIT7 => #SEN8)
   END_RUNG
   // the same network as SCL:
   "DECODER"(INBYTE := "DATARCVS",
             BIT0 => "SEN1",
             BIT1 => "SEN2",
             BIT2 => "SEN3",
             BIT3 => "SEN4",
             BIT4 => "SEN5",
             BIT5 => #SEN6,
             BIT6 => #SEN7,
             BIT7 => #SEN8);
END_REGION

REGION Network 8
   "TRCV_CONTROL_COUNTER"(EN_R := "Clock_10Hz",   // TRCV_C
                          CONT := TRUE,
                          CONNECT := "_01_CONTROL_Receive_DB_1",
                          DATA := "COUNT1");
END_REGION

REGION Network 9
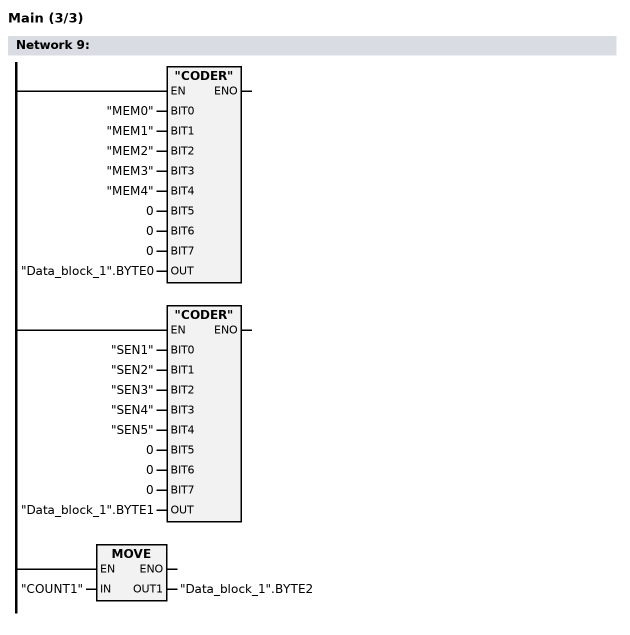
   RUNG wire#powerrail
      "CODER"(BIT0 := "MEM0", BIT1 := "MEM1", BIT2 := "MEM2", BIT3 := "MEM3", BIT4 := "MEM4", BIT5 := 0, BIT6 := 0, BIT7 := 0, OUT := "Data_block_1".BYTE0)
   END_RUNG
   RUNG wire#powerrail
      "CODER"(BIT0 := "SEN1", BIT1 := "SEN2", BIT2 := "SEN3", BIT3 := "SEN4", BIT4 := "SEN5", BIT5 := 0, BIT6 := 0, BIT7 := 0, OUT := "Data_block_1".BYTE1)
   END_RUNG
   RUNG wire#powerrail
      Move(in := "COUNT1", out1 => "Data_block_1".BYTE2)
   END_RUNG
   // the same network as SCL:
   "CODER"(BIT0 := "MEM0",
           BIT1 := "MEM1",
           BIT2 := "MEM2",
           BIT3 := "MEM3",
           BIT4 := "MEM4",
           BIT5 := 0,
           BIT6 := 0,
           BIT7 := 0,
           OUT := "Data_block_1".BYTE0);
   "CODER"(BIT0 := "SEN1",
           BIT1 := "SEN2",
           BIT2 := "SEN3",
           BIT3 := "SEN4",
           BIT4 := "SEN5",
           BIT5 := 0,
           BIT6 := 0,
           BIT7 := 0,
           OUT := "Data_block_1".BYTE1);
   "Data_block_1".BYTE2 := "COUNT1";
END_REGION
END_ORGANIZATION_BLOCK

// ===== PLC "02_ALMACEN"  CPU 1214C AC/DC/Rly =====

VAR_GLOBAL   // PLC tag table "Default tag table"
   "START" AT %I8.1 : Bool;
   "STOP" AT %I8.3 : Bool;
   "SEN1" AT %I1.5 : Bool;
   "SEN2" AT %I1.4 : Bool;
   "SEN3" AT %I8.0 : Bool;
   "BIT0XIN" AT %I0.0 : Bool;
   "BIT1XIN" AT %I0.1 : Bool;
   "BIT2XIN" AT %I0.2 : Bool;
   "BIT3XIN" AT %I0.3 : Bool;
   "BUSYX" AT %I1.0 : Bool;
   "BIT0YIN" AT %I0.4 : Bool;
   "BIT1YIN" AT %I0.5 : Bool;
   "BIT2YIN" AT %I0.6 : Bool;
   "BIT3YIN" AT %I0.7 : Bool;
   "BUSYY" AT %I1.2 : Bool;
   "BIT0XOUT" AT %Q0.0 : Bool;
   "BIT1XOUT" AT %Q0.1 : Bool;
   "BIT2XOUT" AT %Q0.2 : Bool;
   "BIT3XOUT" AT %Q0.3 : Bool;
   "RESETXY" AT %Q1.0 : Bool;
   "BIT0YOUT" AT %Q0.4 : Bool;
   "BIT1YOUT" AT %Q0.5 : Bool;
   "BIT2YOUT" AT %Q0.6 : Bool;
   "BIT3YOUT" AT %Q0.7 : Bool;
   "STOPXY" AT %Q1.1 : Bool;
   "VALVEZ" AT %Q8.0 : Bool;
   "PINZA" AT %Q8.1 : Bool;
   "ALARM" AT %Q8.3 : Bool;
   "MEM0" AT %M0.0 : Bool;
   "MEM1" AT %M0.1 : Bool;
   "MEM2" AT %M0.2 : Bool;
   "MEM3" AT %M0.3 : Bool;
   "MEM4" AT %M0.4 : Bool;
   "MEM5" AT %M0.5 : Bool;
   "MEM6" AT %M0.6 : Bool;
   "MEM7" AT %M0.7 : Bool;
   "MEM8" AT %M1.0 : Bool;
   "MEM9" AT %M1.1 : Bool;
   "MEM10" AT %M1.2 : Bool;
   "MEM11" AT %M1.3 : Bool;
   "MEM12" AT %M1.4 : Bool;
   "VALXIN" AT %MW5 : Int;
   "VALXOUT" AT %MW8 : Int;
   "VALYIN" AT %MW10 : Int;
   "VALYOUT" AT %MW12 : Int;
   "System_Byte" AT %MB1001 : Byte;
   "FirstScan" AT %M1001.0 : Bool;
   "DiagStatusUpdate" AT %M1001.1 : Bool;
   "AlwaysTRUE" AT %M1001.2 : Bool;
   "AlwaysFALSE" AT %M1001.3 : Bool;
   "Clock_Byte" AT %MB1000 : Byte;
   "Clock_10Hz" AT %M1000.0 : Bool;
   "Clock_5Hz" AT %M1000.1 : Bool;
   "Clock_2.5Hz" AT %M1000.2 : Bool;
   "Clock_2Hz" AT %M1000.3 : Bool;
   "Clock_1.25Hz" AT %M1000.4 : Bool;
   "Clock_1Hz" AT %M1000.5 : Bool;
   "Clock_0.625Hz" AT %M1000.6 : Bool;
   "Clock_0.5Hz" AT %M1000.7 : Bool;
   "MEMREST" AT %M1.5 : Bool;
   "MEMYP" AT %M1.6 : Bool;
   "MEMYO" AT %M1.7 : Bool;
   "BYTE2SEND" AT %MB2 : Byte;
   "ENDPROCESS" AT %M3.0 : Bool;
   "FIN" AT %M3.1 : Bool;
   "STATUS2SEND" AT %M3.2 : Bool;
   "BYTEINST" AT %MB4 : Byte;
   "STATES" AT %M3.3 : Bool;
   "MEMNEW" AT %M3.4 : Bool;
   "MEMYP2" AT %M3.5 : Bool;
   "MEMYO2" AT %M3.6 : Bool;
   "VALYOUT2F" AT %MW14 : Int;
   "MEMAUX1" AT %M3.7 : Bool;
   "ME0" AT %M7.0 : Bool;
   "VALX" AT %MW16 : Int;
   "VALY" AT %MW18 : Int;
   "SSUBS" AT %M7.1 : Bool;
   "SADD" AT %M7.2 : Bool;
   "STATE1" AT %M7.3 : Bool;
   "STATE2" AT %M7.4 : Bool;
   "TRIGADD" AT %M7.5 : Bool;
   "TRIGSUBADD" AT %M7.6 : Bool;
   "TRIGFUNC" AT %M7.7 : Bool;
   "TRIGFUNC2" AT %M20.0 : Bool;
   "TRIGORIGIN" AT %M20.1 : Bool;
   "TRIGORIGIN2" AT %M20.2 : Bool;
   "MEMORIGIN" AT %M20.3 : Bool;
   "MORIGIN" AT %M20.4 : Bool;
   "MEMENABLE" AT %M20.5 : Bool;
   "AUTOMODE" AT %I8.2 : Bool;
   "MEMAUX2" AT %M20.6 : Bool;
END_VAR

// folder: System blocks/Program resources

DATA_BLOCK "TIMER2"   // DB1
{ S7_Optimized_Access := 'TRUE' }
AUTHOR : Simatic
FAMILY : IEC
NAME : IEC_TMR
VERSION : 1.0
// stored: InstanceOfName IEC_TIMER
"IEC_TIMER"
BEGIN
END_DATA_BLOCK

DATA_BLOCK "TIMER1"   // DB2
{ S7_Optimized_Access := 'TRUE' }
AUTHOR : Simatic
FAMILY : IEC
NAME : IEC_TMR
VERSION : 1.0
// stored: InstanceOfName IEC_TIMER
"IEC_TIMER"
BEGIN
END_DATA_BLOCK

DATA_BLOCK "TIMER3"   // DB3
{ S7_Optimized_Access := 'TRUE' }
AUTHOR : Simatic
FAMILY : IEC
NAME : IEC_TMR
VERSION : 1.0
// stored: InstanceOfName IEC_TIMER
"IEC_TIMER"
BEGIN
END_DATA_BLOCK

DATA_BLOCK "_02_ALMACEN_Receive_DB"   // DB4
{ S7_Optimized_Access := 'TRUE' }
AUTHOR : SIMATIC
FAMILY : MC7Plus
NAME : TC_IP_v4
VERSION : 1.0
// stored: InstanceOfName TCON_IP_v4
"TCON_IP_v4"
BEGIN
   ID := 1;
   InterfaceId := 64;
   LocalPort := 2000;
   RemoteAddress.ADDR[1] := 192;
   RemoteAddress.ADDR[2] := 168;
   RemoteAddress.ADDR[4] := 3;
END_DATA_BLOCK

DATA_BLOCK "_02_ALMACEN_Send_DB"   // DB6
{ S7_Optimized_Access := 'TRUE' }
AUTHOR : SIMATIC
FAMILY : MC7Plus
NAME : TC_IP_v4
VERSION : 1.0
// stored: InstanceOfName TCON_IP_v4
"TCON_IP_v4"
BEGIN
   ID := 5;
   InterfaceId := 64;
   RemotePort := 2000;
   ActiveEstablished := true;
   RemoteAddress.ADDR[1] := 192;
   RemoteAddress.ADDR[2] := 168;
   RemoteAddress.ADDR[4] := 3;
END_DATA_BLOCK

// folder: (top level)

FUNCTION "DecToBin" : Void   // FC1, FBD
{ S7_Optimized_Access := 'TRUE' }
VERSION : 0.1
   VAR_INPUT
      dec : Int;
   END_VAR
   VAR_OUTPUT
      bit0 : Bool;
      bit1 : Bool;
      bit2 : Bool;
      bit3 : Bool;
   END_VAR
   VAR_TEMP
      secdec : Int;
      thirdec : Int;
      quardec : Int;
      bit0s : Int;
      bit1s : Int;
      bit2s : Int;
      bit3s : Int;
   END_VAR
BEGIN

REGION Network 1
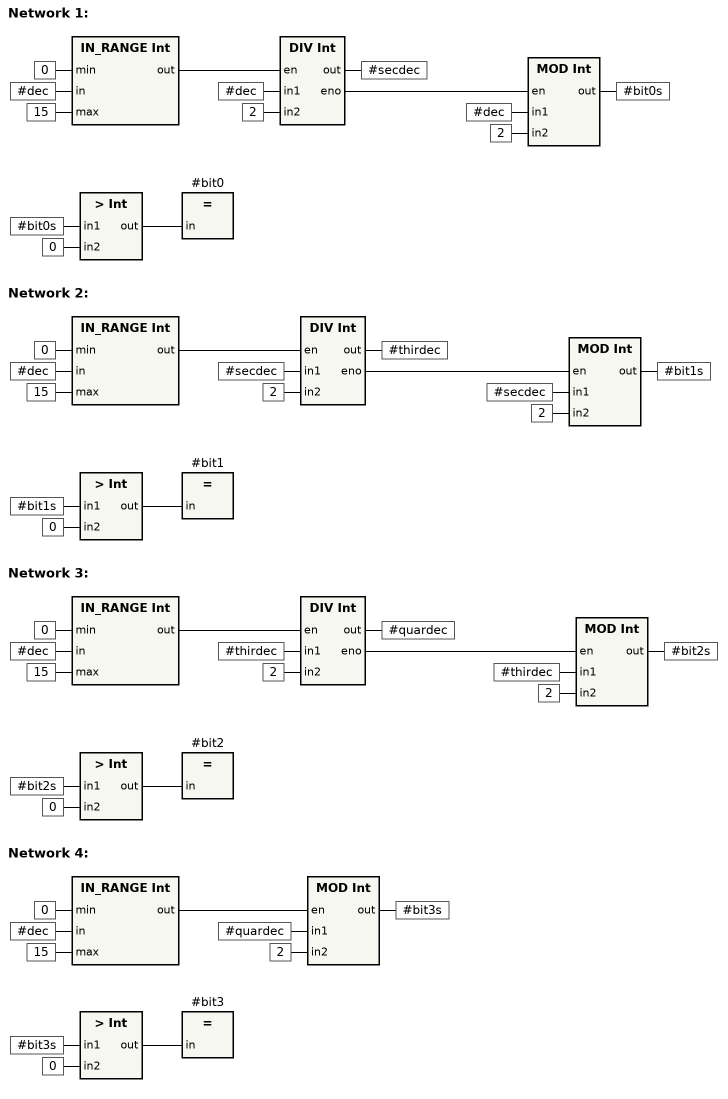
   IF (0 <= #dec) AND (#dec <= 15) THEN
       #secdec := #dec / 2;
       #bit0s := #dec MOD 2;
   END_IF;
   #bit0 := #bit0s > 0;
END_REGION

REGION Network 2
   IF (0 <= #dec) AND (#dec <= 15) THEN
       #thirdec := #secdec / 2;
       #bit1s := #secdec MOD 2;
   END_IF;
   #bit1 := #bit1s > 0;
END_REGION

REGION Network 3
   IF (0 <= #dec) AND (#dec <= 15) THEN
       #quardec := #thirdec / 2;
       #bit2s := #thirdec MOD 2;
   END_IF;
   #bit2 := #bit2s > 0;
END_REGION

REGION Network 4
   IF (0 <= #dec) AND (#dec <= 15) THEN #bit3s := #quardec MOD 2; END_IF;
   #bit3 := #bit3s > 0;
END_REGION
END_FUNCTION

FUNCTION "BinToDec" : Void   // FC2, FBD
{ S7_Optimized_Access := 'TRUE' }
VERSION : 0.1
   VAR_INPUT
      bit0 : Bool;
      bit1 : Bool;
      bit2 : Bool;
      bit3 : Bool;
   END_VAR
   VAR_OUTPUT
      decimal : Int;
   END_VAR
   VAR_TEMP
      dec0 : Int;
      dec1 : Int;
      dec2 : Int;
      dec3 : Int;
   END_VAR
BEGIN

REGION Network 1
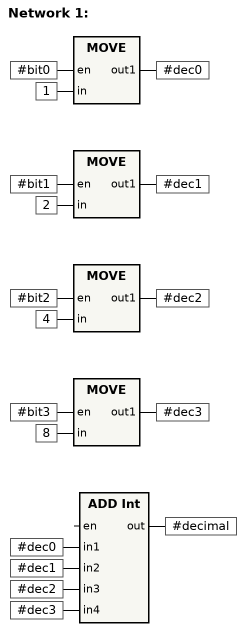
   IF #bit0 THEN #dec0 := 1; END_IF;
   IF #bit1 THEN #dec1 := 2; END_IF;
   IF #bit2 THEN #dec2 := 4; END_IF;
   IF #bit3 THEN #dec3 := 8; END_IF;
   #decimal := #dec0 + #dec1 + #dec2 + #dec3;
END_REGION
END_FUNCTION

FUNCTION "CODER" : Void   // FC3, FBD
{ S7_Optimized_Access := 'TRUE' }
VERSION : 0.1
   VAR_INPUT
      BIT0 : Bool;
      BIT1 : Bool;
      BIT2 : Bool;
      BIT3 : Bool;
      BIT4 : Bool;
      BIT5 : Bool;
      BIT6 : Bool;
      BIT7 : Bool;
   END_VAR
   VAR_IN_OUT
      OUT : Byte;
   END_VAR
   VAR_TEMP
      MASK0 : Byte;
      MASK1 : Byte;
      MASK2 : Byte;
      MASK3 : Byte;
      MASK4 : Byte;
      MASK5 : Byte;
      MASK6 : Byte;
      MASK7 : Byte;
      MASK : Byte;
      MASK0N : Byte;
      MASK1N : Byte;
      MASK2N : Byte;
      MASK3N : Byte;
      MASK4N : Byte;
      MASK5N : Byte;
      MASK6N : Byte;
      MASK7N : Byte;
      MASKN : Byte;
   END_VAR
BEGIN

REGION Network 1
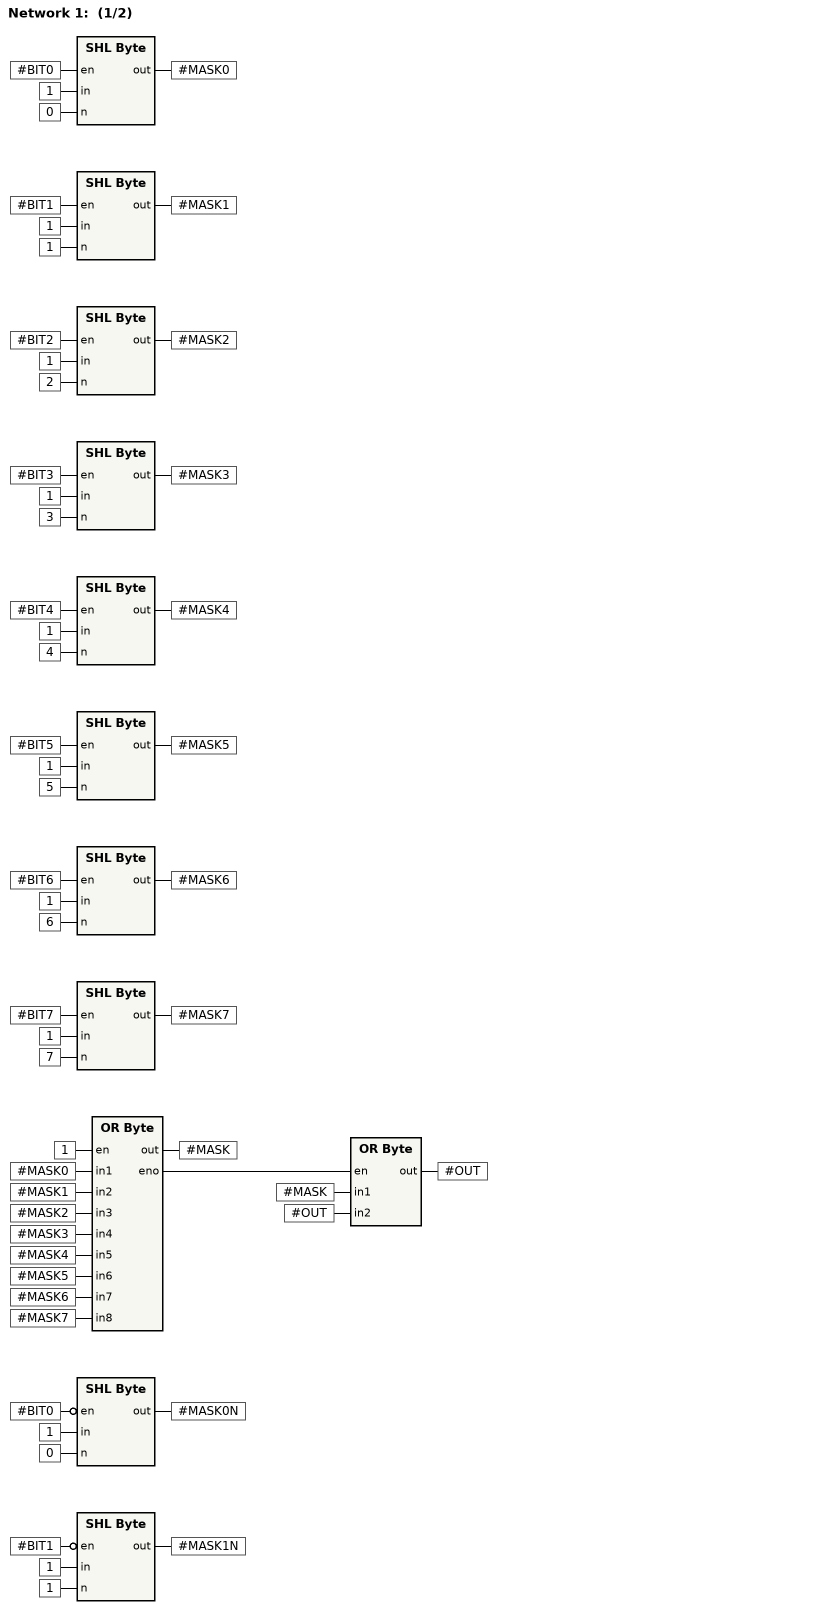
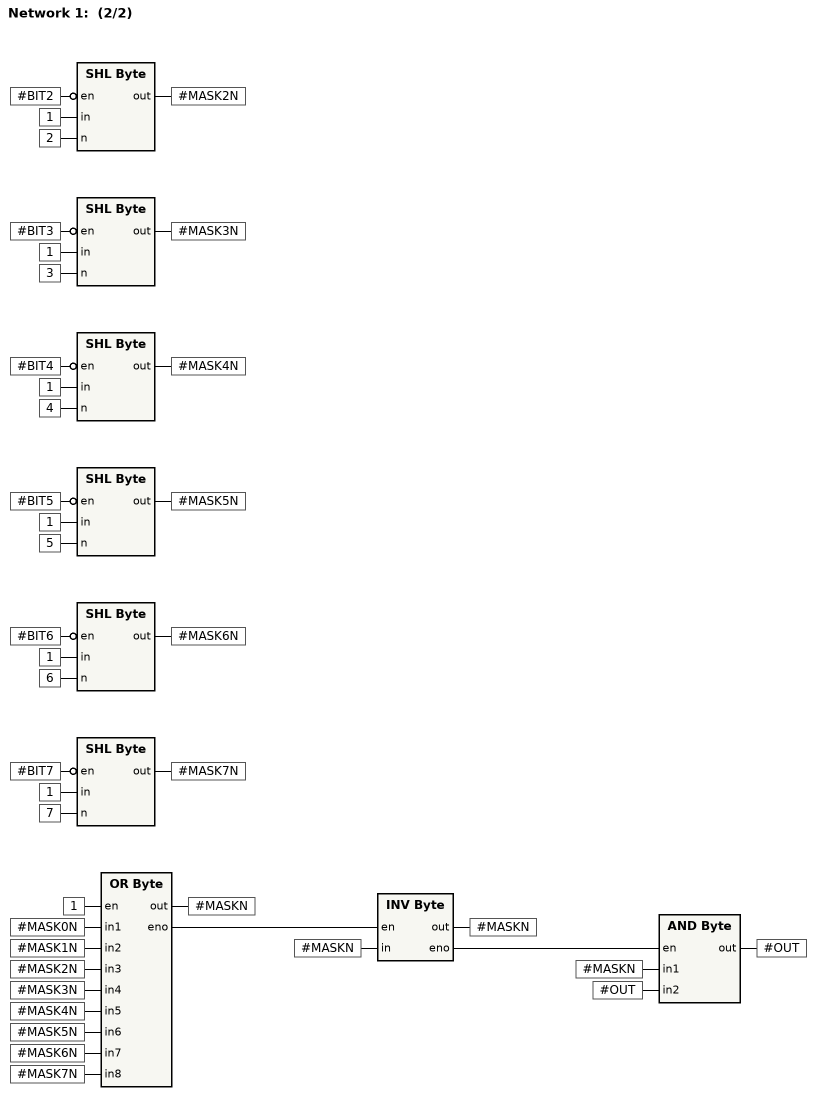
   IF #BIT0 THEN #MASK0 := SHL(IN := 1, N := 0); END_IF;
   IF #BIT1 THEN #MASK1 := SHL(IN := 1, N := 1); END_IF;
   IF #BIT2 THEN #MASK2 := SHL(IN := 1, N := 2); END_IF;
   IF #BIT3 THEN #MASK3 := SHL(IN := 1, N := 3); END_IF;
   IF #BIT4 THEN #MASK4 := SHL(IN := 1, N := 4); END_IF;
   IF #BIT5 THEN #MASK5 := SHL(IN := 1, N := 5); END_IF;
   IF #BIT6 THEN #MASK6 := SHL(IN := 1, N := 6); END_IF;
   IF #BIT7 THEN #MASK7 := SHL(IN := 1, N := 7); END_IF;
   IF 1 THEN
       #MASK := #MASK0 OR #MASK1 OR #MASK2 OR #MASK3 OR #MASK4 OR #MASK5 OR #MASK6 OR #MASK7;
       #OUT := #MASK OR #OUT;
   END_IF;
   IF NOT #BIT0 THEN #MASK0N := SHL(IN := 1, N := 0); END_IF;
   IF NOT #BIT1 THEN #MASK1N := SHL(IN := 1, N := 1); END_IF;
   IF NOT #BIT2 THEN #MASK2N := SHL(IN := 1, N := 2); END_IF;
   IF NOT #BIT3 THEN #MASK3N := SHL(IN := 1, N := 3); END_IF;
   IF NOT #BIT4 THEN #MASK4N := SHL(IN := 1, N := 4); END_IF;
   IF NOT #BIT5 THEN #MASK5N := SHL(IN := 1, N := 5); END_IF;
   IF NOT #BIT6 THEN #MASK6N := SHL(IN := 1, N := 6); END_IF;
   IF NOT #BIT7 THEN #MASK7N := SHL(IN := 1, N := 7); END_IF;
   IF 1 THEN
       #MASKN := #MASK0N OR #MASK1N OR #MASK2N OR #MASK3N OR #MASK4N OR #MASK5N OR #MASK6N OR #MASK7N;
       #MASKN := NOT #MASKN;
       #OUT := #MASKN AND #OUT;
   END_IF;
END_REGION
END_FUNCTION

FUNCTION "DECODER" : Void   // FC4, FBD
{ S7_Optimized_Access := 'TRUE' }
VERSION : 0.1
   VAR_INPUT
      INBYTE : Byte;
   END_VAR
   VAR_OUTPUT
      BIT0 : Bool;
      BIT1 : Bool;
      BIT2 : Bool;
      BIT3 : Bool;
      BIT4 : Bool;
      BIT5 : Bool;
      BIT6 : Bool;
      BIT7 : Bool;
   END_VAR
   VAR_TEMP
      MASK0 : Byte;
      MASK1 : Byte;
      MASK2 : Byte;
      MASK3 : Byte;
      MASK4 : Byte;
      MASK5 : Byte;
      MASK6 : Byte;
      MASK7 : Byte;
      OUTBIT0 : Byte;
      OUTBIT1 : Byte;
      OUTBIT2 : Byte;
      OUTBIT3 : Byte;
      OUTBIT4 : Byte;
      OUTBIT5 : Byte;
      OUTBIT6 : Byte;
      OUTBIT7 : Byte;
   END_VAR
BEGIN

REGION Network 1
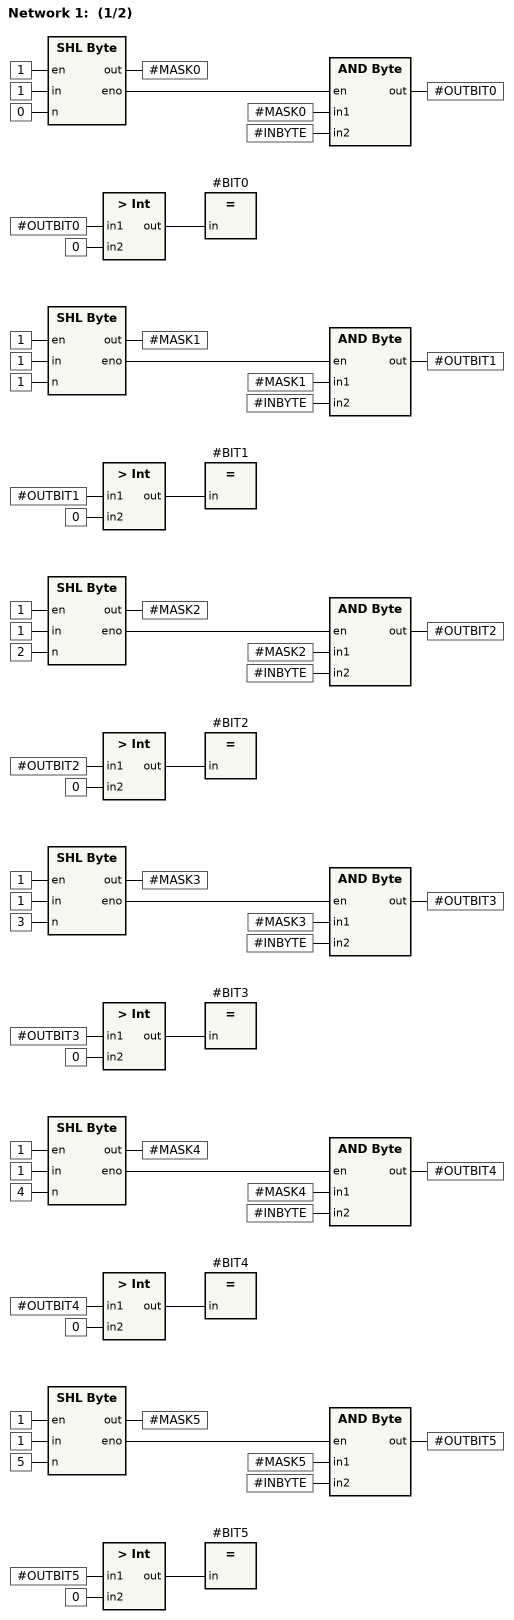
